LIN {X 0,Y 249.344,Z 174.923,A -85,B 0,C 180,E1 -18909.737,E2 -18909.737} C_VEL
LIN {X 0,Y 249.206,Z 174.945,A -85,B 0,C 180,E1 -18914.703,E2 -18914.703} C_VEL
LIN {X 0,Y 249.14,Z 174.944,A -85,B 0,C 180,E1 -18918.077,E2 -18918.077} C_VEL
LIN {X 0,Y 249.088,Z 174.954,A -85,B 0,C 180,E1 -18921.518,E2 -18921.518} C_VEL
LIN {X 0,Y 249.131,Z 174.951,A -85,B 0,C 180,E1 -18925.482,E2 -18925.482} C_VEL
LIN {X 0,Y 249.084,Z 174.957,A -85,B 0,C 180,E1 -18928.994,E2 -18928.994} C_VEL
LIN {X 0,Y 249.037,Z 174.96,A -85,B 0,C 180,E1 -18932.425,E2 -18932.425} C_VEL
LIN {X 0,Y 249.07,Z 174.957,A -85,B 0,C 180,E1 -18936.339,E2 -18936.339} C_VEL
LIN {X 0,Y 249.027,Z 174.966,A -85,B 0,C 180,E1 -18940.474,E2 -18940.474} C_VEL
LIN {X 0,Y 249.003,Z 174.965,A -85,B 0,C 180,E1 -18944.879,E2 -18944.879} C_VEL
LIN {X 0,Y 249.017,Z 174.965,A -85,B 0,C 180,E1 -18947.363,E2 -18947.363} C_VEL
LIN {X 0,Y 249.046,Z 174.962,A -85,B 0,C 180,E1 -18952.2,E2 -18952.2} C_VEL
LIN {X 0,Y 249.103,Z 175.108,A -85,B 0,C 180,E1 -18955.468,E2 -18955.468} C_VEL
LIN {X 0,Y 249.854,Z 178.125,A -85,B 0,C 180,E1 -18956.815,E2 -18956.815} C_VEL
LIN {X 0,Y 259.148,Z 197.045,A -85,B 0,C 180,E1 -18958.762,E2 -18958.762} C_VEL
LIN {X 0,Y 265.414,Z 211.933,A -85,B 0,C 180,E1 -18960.042,E2 -18960.042} C_VEL
LIN {X 0,Y 267.439,Z 217.922,A -85,B 0,C 180,E1 -18960.475,E2 -18960.475} C_VEL
LIN {X 0,Y 265.215,Z 283.423,A -85,B 0,C 180,E1 -18962.211,E2 -18962.211} C_VEL
LIN {X 0,Y 264.278,Z 296.661,A -85,B 0,C 180,E1 -18962.802,E2 -18962.802} C_VEL
LIN {X 0,Y 262.847,Z 309.804,A -85,B 0,C 180,E1 -18963.714,E2 -18963.714} C_VEL
LIN {X 0,Y 261.114,Z 322.253,A -85,B 0,C 180,E1 -18964.918,E2 -18964.918} C_VEL
LIN {X 0,Y 259.054,Z 333.896,A -85,B 0,C 180,E1 -18966.412,E2 -18966.412} C_VEL
LIN {X 0,Y 256.908,Z 344.67,A -85,B 0,C 180,E1 -18968.179,E2 -18968.179} C_VEL
LIN {X 0,Y 254.989,Z 354.577,A -85,B 0,C 180,E1 -18970.267,E2 -18970.267} C_VEL
LIN {X 0,Y 252.694,Z 363.495,A -85,B 0,C 180,E1 -18972.604,E2 -18972.604} C_VEL
LIN {X 0,Y 250.914,Z 370.67,A -85,B 0,C 180,E1 -18974.984,E2 -18974.984} C_VEL
LIN {X 0,Y 249.694,Z 375.507,A -85,B 0,C 180,E1 -18976.987,E2 -18976.987} C_VEL
LIN {X 0,Y 248.535,Z 380.207,A -85,B 0,C 180,E1 -18979.409,E2 -18979.409} C_VEL
LIN {X 0,Y 247.828,Z 383.8,A -85,B 0,C 180,E1 -18981.848,E2 -18981.848} C_VEL
LIN {X 0,Y 247.377,Z 386.053,A -85,B 0,C 180,E1 -18983.911,E2 -18983.911} C_VEL
LIN {X 0,Y 247.078,Z 388.044,A -85,B 0,C 180,E1 -18986.739,E2 -18986.739} C_VEL
LIN {X 0,Y 246.944,Z 388.884,A -85,B 0,C 180,E1 -18990,E2 -18990} C_VEL
LIN {X 0,Y 246.971,Z 388.691,A -85,B 0,C 180,E1 -18991.631,E2 -18991.631} C_VEL
LIN {X 0,Y 247.075,Z 388.104,A -85,B 0,C 180,E1 -18993.261,E2 -18993.261} C_VEL
LIN {X 0,Y 247.393,Z 385.779,A -85,B 0,C 180,E1 -18996.525,E2 -18996.525} C_VEL
LIN {X 0,Y 247.985,Z 382.908,A -85,B 0,C 180,E1 -18998.967,E2 -18998.967} C_VEL
LIN {X 0,Y 248.859,Z 379.014,A -85,B 0,C 180,E1 -19001.402,E2 -19001.402} C_VEL
LIN {X 0,Y 250.108,Z 373.989,A -85,B 0,C 180,E1 -19003.818,E2 -19003.818} C_VEL
LIN {X 0,Y 251.645,Z 367.662,A -85,B 0,C 180,E1 -19006.217,E2 -19006.217} C_VEL
LIN {X 0,Y 253.716,Z 359.739,A -85,B 0,C 180,E1 -19008.575,E2 -19008.575} C_VEL
LIN {X 0,Y 255.61,Z 351.261,A -85,B 0,C 180,E1 -19010.618,E2 -19010.618} C_VEL
LIN {X 0,Y 257.585,Z 341.814,A -85,B 0,C 180,E1 -19012.456,E2 -19012.456} C_VEL
LIN {X 0,Y 259.734,Z 330.721,A -85,B 0,C 180,E1 -19014.158,E2 -19014.158} C_VEL
LIN {X 0,Y 261.56,Z 319.844,A -85,B 0,C 180,E1 -19015.462,E2 -19015.462} C_VEL
LIN {X 0,Y 263.224,Z 307.822,A -85,B 0,C 180,E1 -19016.565,E2 -19016.565} C_VEL
LIN {X 0,Y 264.419,Z 295.46,A -85,B 0,C 180,E1 -19017.397,E2 -19017.397} C_VEL
LIN {X 0,Y 265.365,Z 282.621,A -85,B 0,C 180,E1 -19017.933,E2 -19017.933} C_VEL
LIN {X 0,Y 267.467,Z 217.517,A -85,B 0,C 180,E1 -19019.667,E2 -19019.667} C_VEL
LIN {X 0,Y 260.917,Z 200.918,A -85,B 0,C 180,E1 -19021.016,E2 -19021.016} C_VEL
LIN {X 0,Y 253.203,Z 184.855,A -85,B 0,C 180,E1 -19022.606,E2 -19022.606} C_VEL
LIN {X 0,Y 249.816,Z 177.906,A -85,B 0,C 180,E1 -19023.394,E2 -19023.394} C_VEL
LIN {X 0,Y 249.057,Z 174.953,A -85,B 0,C 180,E1 -19024.827,E2 -19024.827} C_VEL
LIN {X 0,Y 249.026,Z 174.967,A -85,B 0,C 180,E1 -19028.38,E2 -19028.38} C_VEL
LIN {X 0,Y 249.01,Z 174.968,A -85,B 0,C 180,E1 -19032.792,E2 -19032.792} C_VEL
LIN {X 0,Y 249.016,Z 174.965,A -85,B 0,C 180,E1 -19037.363,E2 -19037.363} C_VEL
LIN {X 0,Y 249.037,Z 174.959,A -85,B 0,C 180,E1 -19041.621,E2 -19041.621} C_VEL
LIN {X 0,Y 249.058,Z 174.956,A -85,B 0,C 180,E1 -19045.641,E2 -19045.641} C_VEL
LIN {X 0,Y 249.052,Z 174.962,A -85,B 0,C 180,E1 -19049.473,E2 -19049.473} C_VEL
LIN {X 0,Y 249.074,Z 174.953,A -85,B 0,C 180,E1 -19053.162,E2 -19053.162} C_VEL
LIN {X 0,Y 249.079,Z 174.954,A -85,B 0,C 180,E1 -19056.732,E2 -19056.732} C_VEL
LIN {X 0,Y 249.111,Z 174.953,A -85,B 0,C 180,E1 -19060.211,E2 -19060.211} C_VEL
LIN {X 0,Y 249.242,Z 174.927,A -85,B 0,C 180,E1 -19063.622,E2 -19063.622} C_VEL
LIN {X 0,Y 249.253,Z 174.937,A -85,B 0,C 180,E1 -19068.616,E2 -19068.616} C_VEL
LIN {X 0,Y 249.479,Z 174.897,A -85,B 0,C 180,E1 -19071.903,E2 -19071.903} C_VEL
LIN {X 0,Y 249.436,Z 174.911,A -85,B 0,C 180,E1 -19076.77,E2 -19076.77} C_VEL
LIN {X 0,Y 249.721,Z 174.87,A -85,B 0,C 180,E1 -19080,E2 -19080} C_VEL
LIN {X 0,Y 249.435,Z 174.912,A -85,B 0,C 180,E1 -19083.23,E2 -19083.23} C_VEL
LIN {X 0,Y 249.379,Z 174.907,A -85,B 0,C 180,E1 -19085.901,E2 -19085.901} C_VEL
LIN {X 0,Y 248.797,Z 174.987,A -85,B 0,C 180,E1 -19087.249,E2 -19087.249} C_VEL
LIN {X 0,Y 247.192,Z 175.192,A -85,B 0,C 180,E1 -19088.57,E2 -19088.57} C_VEL
LIN {X 0,Y 243.31,Z 175.672,A -85,B 0,C 180,E1 -19091.228,E2 -19091.228} C_VEL
LIN {X 0,Y 242.229,Z 175.8,A -85,B 0,C 180,E1 -19092.619,E2 -19092.619} C_VEL
LIN {X 0,Y 242.153,Z 175.807,A -85,B 0,C 180,E1 -19093.091,E2 -19093.091} C_VEL
LIN {X 0,Y 242.15,Z 175.819,A -85,B 0,C 180,E1 -19096.872,E2 -19096.872} C_VEL
LIN {X 0,Y 242.026,Z 175.834,A -85,B 0,C 180,E1 -19101.687,E2 -19101.687} C_VEL
LIN {X 0,Y 242.066,Z 175.824,A -85,B 0,C 180,E1 -19105.838,E2 -19105.838} C_VEL
LIN {X 0,Y 242.007,Z 175.835,A -85,B 0,C 180,E1 -19109.583,E2 -19109.583} C_VEL
LIN {X 0,Y 241.98,Z 175.841,A -85,B 0,C 180,E1 -19113.493,E2 -19113.493} C_VEL
LIN {X 0,Y 241.989,Z 175.839,A -85,B 0,C 180,E1 -19117.582,E2 -19117.582} C_VEL
LIN {X 0,Y 241.933,Z 175.846,A -85,B 0,C 180,E1 -19121.923,E2 -19121.923} C_VEL
LIN {X 0,Y 241.92,Z 175.85,A -85,B 0,C 180,E1 -19126.575,E2 -19126.575} C_VEL
LIN {X 0,Y 241.972,Z 176.038,A -85,B 0,C 180,E1 -19130.843,E2 -19130.843} C_VEL
LIN {X 0,Y 244.268,Z 184.837,A -85,B 0,C 180,E1 -19134.87,E2 -19134.87} C_VEL
LIN {X 0,Y 244.871,Z 187.317,A -85,B 0,C 180,E1 -19135.941,E2 -19135.941} C_VEL
LIN {X 0,Y 253.51,Z 206.311,A -85,B 0,C 180,E1 -19137.867,E2 -19137.867} C_VEL
LIN {X 0,Y 257.423,Z 216.174,A -85,B 0,C 180,E1 -19138.725,E2 -19138.725} C_VEL
LIN {X 0,Y 260.42,Z 235.313,A -85,B 0,C 180,E1 -19139.722,E2 -19139.722} C_VEL
LIN {X 0,Y 260.581,Z 240.387,A -85,B 0,C 180,E1 -19139.901,E2 -19139.901} C_VEL
LIN {X 0,Y 258.581,Z 296.119,A -85,B 0,C 180,E1 -19141.433,E2 -19141.433} C_VEL
LIN {X 0,Y 257.413,Z 309.243,A -85,B 0,C 180,E1 -19142.069,E2 -19142.069} C_VEL
LIN {X 0,Y 255.916,Z 321.325,A -85,B 0,C 180,E1 -19142.945,E2 -19142.945} C_VEL
LIN {X 0,Y 253.998,Z 333.525,A -85,B 0,C 180,E1 -19144.164,E2 -19144.164} C_VEL
LIN {X 0,Y 251.737,Z 345.085,A -85,B 0,C 180,E1 -19145.683,E2 -19145.683} C_VEL
LIN {X 0,Y 249.416,Z 355.496,A -85,B 0,C 180,E1 -19147.423,E2 -19147.423} C_VEL
LIN {X 0,Y 247.472,Z 364.011,A -85,B 0,C 180,E1 -19149.207,E2 -19149.207} C_VEL
LIN {X 0,Y 245.32,Z 373.244,A -85,B 0,C 180,E1 -19151.631,E2 -19151.631} C_VEL
LIN {X 0,Y 243.415,Z 380.664,A -85,B 0,C 180,E1 -19154.081,E2 -19154.081} C_VEL
LIN {X 0,Y 241.865,Z 386.623,A -85,B 0,C 180,E1 -19156.558,E2 -19156.558} C_VEL
LIN {X 0,Y 240.87,Z 391.336,A -85,B 0,C 180,E1 -19159.068,E2 -19159.068} C_VEL
LIN {X 0,Y 240.211,Z 394.938,A -85,B 0,C 180,E1 -19161.588,E2 -19161.588} C_VEL
LIN {X 0,Y 239.926,Z 396.795,A -85,B 0,C 180,E1 -19163.271,E2 -19163.271} C_VEL
LIN {X 0,Y 239.755,Z 399.185,A -85,B 0,C 180,E1 -19166.639,E2 -19166.639} C_VEL
LIN {X 0,Y 239.808,Z 399.793,A -85,B 0,C 180,E1 -19168.321,E2 -19168.321} C_VEL
LIN {X 0,Y 239.846,Z 400.005,A -85,B 0,C 180,E1 -19170,E2 -19170} C_VEL
LIN {X 0,Y 239.808,Z 399.782,A -85,B 0,C 180,E1 -19171.679,E2 -19171.679} C_VEL
LIN {X 0,Y 239.771,Z 398.373,A -85,B 0,C 180,E1 -19174.736,E2 -19174.736} C_VEL
LIN {X 0,Y 239.926,Z 396.76,A -85,B 0,C 180,E1 -19176.729,E2 -19176.729} C_VEL
LIN {X 0,Y 240.387,Z 393.815,A -85,B 0,C 180,E1 -19179.253,E2 -19179.253} C_VEL
LIN {X 0,Y 241.188,Z 389.833,A -85,B 0,C 180,E1 -19181.769,E2 -19181.769} C_VEL
LIN {X 0,Y 242.6,Z 383.713,A -85,B 0,C 180,E1 -19184.684,E2 -19184.684} C_VEL
LIN {X 0,Y 244.335,Z 377.034,A -85,B 0,C 180,E1 -19187.147,E2 -19187.147} C_VEL
LIN {X 0,Y 246.353,Z 368.317,A -85,B 0,C 180,E1 -19189.707,E2 -19189.707} C_VEL
LIN {X 0,Y 248.269,Z 360.245,A -85,B 0,C 180,E1 -19191.593,E2 -19191.593} C_VEL
LIN {X 0,Y 250.662,Z 349.747,A -85,B 0,C 180,E1 -19193.549,E2 -19193.549} C_VEL
LIN {X 0,Y 253.102,Z 337.93,A -85,B 0,C 180,E1 -19195.272,E2 -19195.272} C_VEL
LIN {X 0,Y 255.057,Z 326.019,A -85,B 0,C 180,E1 -19196.6,E2 -19196.6} C_VEL
LIN {X 0,Y 256.788,Z 313.622,A -85,B 0,C 180,E1 -19197.617,E2 -19197.617} C_VEL
LIN {X 0,Y 258.195,Z 300.844,A -85,B 0,C 180,E1 -19198.336,E2 -19198.336} C_VEL
LIN {X 0,Y 258.927,Z 287.293,A -85,B 0,C 180,E1 -19198.802,E2 -19198.802} C_VEL
LIN {X 0,Y 260.493,Z 236.282,A -85,B 0,C 180,E1 -19200.193,E2 -19200.193} C_VEL
LIN {X 0,Y 257.318,Z 215.805,A -85,B 0,C 180,E1 -19201.253,E2 -19201.253} C_VEL
LIN {X 0,Y 250.055,Z 198.58,A -85,B 0,C 180,E1 -19202.835,E2 -19202.835} C_VEL
LIN {X 0,Y 244.825,Z 187.196,A -85,B 0,C 180,E1 -19204.049,E2 -19204.049} C_VEL
LIN {X 0,Y 242.739,Z 178.842,A -85,B 0,C 180,E1 -19207.778,E2 -19207.778} C_VEL
LIN {X 0,Y 241.957,Z 175.847,A -85,B 0,C 180,E1 -19209.252,E2 -19209.252} C_VEL
LIN {X 0,Y 241.921,Z 175.851,A -85,B 0,C 180,E1 -19213.425,E2 -19213.425} C_VEL
LIN {X 0,Y 241.934,Z 175.849,A -85,B 0,C 180,E1 -19218.077,E2 -19218.077} C_VEL
LIN {X 0,Y 241.989,Z 175.842,A -85,B 0,C 180,E1 -19222.418,E2 -19222.418} C_VEL
LIN {X 0,Y 241.979,Z 175.844,A -85,B 0,C 180,E1 -19226.507,E2 -19226.507} C_VEL
LIN {X 0,Y 241.978,Z 175.843,A -85,B 0,C 180,E1 -19230.612,E2 -19230.612} C_VEL
LIN {X 0,Y 242.032,Z 175.836,A -85,B 0,C 180,E1 -19234.179,E2 -19234.179} C_VEL
LIN {X 0,Y 242.026,Z 175.835,A -85,B 0,C 180,E1 -19238.314,E2 -19238.314} C_VEL
LIN {X 0,Y 242.164,Z 175.814,A -85,B 0,C 180,E1 -19243.278,E2 -19243.278} C_VEL
LIN {X 0,Y 242.181,Z 175.812,A -85,B 0,C 180,E1 -19248.28,E2 -19248.28} C_VEL
LIN {X 0,Y 242.401,Z 175.788,A -85,B 0,C 180,E1 -19251.665,E2 -19251.665} C_VEL
LIN {X 0,Y 242.257,Z 175.804,A -85,B 0,C 180,E1 -19255.007,E2 -19255.007} C_VEL
LIN {X 0,Y 242.637,Z 175.756,A -85,B 0,C 180,E1 -19258.34,E2 -19258.34} C_VEL
LIN {X 0,Y 242.636,Z 175.761,A -85,B 0,C 180,E1 -19261.66,E2 -19261.66} C_VEL
LIN {X 0,Y 242.423,Z 175.781,A -85,B 0,C 180,E1 -19266.659,E2 -19266.659} C_VEL
LIN {X 0,Y 242.268,Z 175.804,A -85,B 0,C 180,E1 -19270.024,E2 -19270.024} C_VEL
LIN {X 0,Y 242.167,Z 175.818,A -85,B 0,C 180,E1 -19275.141,E2 -19275.141} C_VEL
LIN {X 0,Y 242.074,Z 175.827,A -85,B 0,C 180,E1 -19278.624,E2 -19278.624} C_VEL
LIN {X 0,Y 242.014,Z 175.833,A -85,B 0,C 180,E1 -19282.18,E2 -19282.18} C_VEL
LIN {X 0,Y 242.067,Z 175.831,A -85,B 0,C 180,E1 -19285.838,E2 -19285.838} C_VEL
LIN {X 0,Y 242.031,Z 175.835,A -85,B 0,C 180,E1 -19289.58,E2 -19289.58} C_VEL
LIN {X 0,Y 241.992,Z 175.84,A -85,B 0,C 180,E1 -19293.491,E2 -19293.491} C_VEL
LIN {X 0,Y 242.003,Z 175.84,A -85,B 0,C 180,E1 -19297.58,E2 -19297.58} C_VEL
LIN {X 0,Y 241.944,Z 175.846,A -85,B 0,C 180,E1 -19301.921,E2 -19301.921} C_VEL
LIN {X 0,Y 241.935,Z 175.847,A -85,B 0,C 180,E1 -19306.571,E2 -19306.571} C_VEL
LIN {X 0,Y 241.958,Z 175.844,A -85,B 0,C 180,E1 -19310.281,E2 -19310.281} C_VEL
LIN {X 0,Y 242.02,Z 175.849,A -85,B 0,C 180,E1 -19314.546,E2 -19314.546} C_VEL
LIN {X 0,Y 242.628,Z 178.345,A -85,B 0,C 180,E1 -19315.691,E2 -19315.691} C_VEL
LIN {X 0,Y 251.925,Z 196.7,A -85,B 0,C 180,E1 -19317.741,E2 -19317.741} C_VEL
LIN {X 0,Y 258.644,Z 212.335,A -85,B 0,C 180,E1 -19319.18,E2 -19319.18} C_VEL
LIN {X 0,Y 261.151,Z 219.015,A -85,B 0,C 180,E1 -19319.719,E2 -19319.719} C_VEL
LIN {X 0,Y 259.029,Z 282.511,A -85,B 0,C 180,E1 -19321.447,E2 -19321.447} C_VEL
LIN {X 0,Y 258.152,Z 295.304,A -85,B 0,C 180,E1 -19321.996,E2 -19321.996} C_VEL
LIN {X 0,Y 256.799,Z 307.717,A -85,B 0,C 180,E1 -19322.826,E2 -19322.826} C_VEL
LIN {X 0,Y 254.972,Z 320.685,A -85,B 0,C 180,E1 -19324.051,E2 -19324.051} C_VEL
LIN {X 0,Y 253.06,Z 331.432,A -85,B 0,C 180,E1 -19325.381,E2 -19325.381} C_VEL
LIN {X 0,Y 250.823,Z 342.491,A -85,B 0,C 180,E1 -19327.144,E2 -19327.144} C_VEL
LIN {X 0,Y 248.865,Z 351.996,A -85,B 0,C 180,E1 -19329.071,E2 -19329.071} C_VEL
LIN {X 0,Y 246.654,Z 360.923,A -85,B 0,C 180,E1 -19331.304,E2 -19331.304} C_VEL
LIN {X 0,Y 244.597,Z 368.613,A -85,B 0,C 180,E1 -19333.731,E2 -19333.731} C_VEL
LIN {X 0,Y 242.762,Z 375.671,A -85,B 0,C 180,E1 -19336.609,E2 -19336.609} C_VEL
LIN {X 0,Y 241.553,Z 380.37,A -85,B 0,C 180,E1 -19339.099,E2 -19339.099} C_VEL
LIN {X 0,Y 240.789,Z 383.963,A -85,B 0,C 180,E1 -19341.608,E2 -19341.608} C_VEL
LIN {X 0,Y 240.287,Z 386.411,A -85,B 0,C 180,E1 -19343.96,E2 -19343.96} C_VEL
LIN {X 0,Y 240.002,Z 388.206,A -85,B 0,C 180,E1 -19346.642,E2 -19346.642} C_VEL
LIN {X 0,Y 239.855,Z 389.046,A -85,B 0,C 180,E1 -19350,E2 -19350} C_VEL
LIN {X 0,Y 239.886,Z 388.853,A -85,B 0,C 180,E1 -19351.679,E2 -19351.679} C_VEL
LIN {X 0,Y 239.997,Z 388.266,A -85,B 0,C 180,E1 -19353.357,E2 -19353.357} C_VEL
LIN {X 0,Y 240.349,Z 385.941,A -85,B 0,C 180,E1 -19356.717,E2 -19356.717} C_VEL
LIN {X 0,Y 240.972,Z 383.069,A -85,B 0,C 180,E1 -19359.23,E2 -19359.23} C_VEL
LIN {X 0,Y 241.897,Z 379.175,A -85,B 0,C 180,E1 -19361.734,E2 -19361.734} C_VEL
LIN {X 0,Y 243.217,Z 374.15,A -85,B 0,C 180,E1 -19364.218,E2 -19364.218} C_VEL
LIN {X 0,Y 244.831,Z 367.822,A -85,B 0,C 180,E1 -19366.682,E2 -19366.682} C_VEL
LIN {X 0,Y 246.999,Z 359.899,A -85,B 0,C 180,E1 -19369.1,E2 -19369.1} C_VEL
LIN {X 0,Y 248.824,Z 352.038,A -85,B 0,C 180,E1 -19371.056,E2 -19371.056} C_VEL
LIN {X 0,Y 251.03,Z 341.973,A -85,B 0,C 180,E1 -19373.076,E2 -19373.076} C_VEL
LIN {X 0,Y 253.291,Z 330.878,A -85,B 0,C 180,E1 -19374.814,E2 -19374.814} C_VEL
LIN {X 0,Y 255.174,Z 320,A -85,B 0,C 180,E1 -19376.147,E2 -19376.147} C_VEL
LIN {X 0,Y 256.908,Z 307.976,A -85,B 0,C 180,E1 -19377.272,E2 -19377.272} C_VEL
LIN {X 0,Y 258.138,Z 295.611,A -85,B 0,C 180,E1 -19378.121,E2 -19378.121} C_VEL
LIN {X 0,Y 259.125,Z 282.763,A -85,B 0,C 180,E1 -19378.667,E2 -19378.667} C_VEL
LIN {X 0,Y 261.284,Z 219.256,A -85,B 0,C 180,E1 -19380.392,E2 -19380.392} C_VEL
LIN {X 0,Y 255.424,Z 204.408,A -85,B 0,C 180,E1 -19381.65,E2 -19381.65} C_VEL
LIN {X 0,Y 248.107,Z 188.989,A -85,B 0,C 180,E1 -19383.225,E2 -19383.225} C_VEL
LIN {X 0,Y 243.691,Z 180.673,A -85,B 0,C 180,E1 -19384.202,E2 -19384.202} C_VEL
LIN {X 0,Y 242.589,Z 178.173,A -85,B 0,C 180,E1 -19384.494,E2 -19384.494} C_VEL
LIN {X 0,Y 242.01,Z 175.835,A -85,B 0,C 180,E1 -19385.666,E2 -19385.666} C_VEL
LIN {X 0,Y 241.957,Z 175.843,A -85,B 0,C 180,E1 -19389.719,E2 -19389.719} C_VEL
LIN {X 0,Y 241.931,Z 175.847,A -85,B 0,C 180,E1 -19394.202,E2 -19394.202} C_VEL
LIN {X 0,Y 241.943,Z 175.843,A -85,B 0,C 180,E1 -19398.079,E2 -19398.079} C_VEL
LIN {X 0,Y 241.999,Z 175.834,A -85,B 0,C 180,E1 -19402.42,E2 -19402.42} C_VEL
LIN {X 0,Y 241.989,Z 175.831,A -85,B 0,C 180,E1 -19406.508,E2 -19406.508} C_VEL
LIN {X 0,Y 242.037,Z 175.831,A -85,B 0,C 180,E1 -19410.587,E2 -19410.587} C_VEL
LIN {X 0,Y 242.068,Z 175.832,A -85,B 0,C 180,E1 -19414.183,E2 -19414.183} C_VEL
LIN {X 0,Y 242.053,Z 175.824,A -85,B 0,C 180,E1 -19418.297,E2 -19418.297} C_VEL
LIN {X 0,Y 242.163,Z 175.811,A -85,B 0,C 180,E1 -19423.278,E2 -19423.278} C_VEL
LIN {X 0,Y 242.186,Z 175.816,A -85,B 0,C 180,E1 -19428.28,E2 -19428.28} C_VEL
LIN {X 0,Y 242.426,Z 175.774,A -85,B 0,C 180,E1 -19431.665,E2 -19431.665} C_VEL
LIN {X 0,Y 242.259,Z 175.81,A -85,B 0,C 180,E1 -19435.007,E2 -19435.007} C_VEL
LIN {X 0,Y 242.636,Z 175.749,A -85,B 0,C 180,E1 -19438.34,E2 -19438.34} C_VEL
LIN {X 0,Y 242.636,Z 175.76,A -85,B 0,C 180,E1 -19441.66,E2 -19441.66} C_VEL
LIN {X 0,Y 242.431,Z 175.774,A -85,B 0,C 180,E1 -19446.659,E2 -19446.659} C_VEL
LIN {X 0,Y 242.314,Z 175.801,A -85,B 0,C 180,E1 -19450.022,E2 -19450.022} C_VEL
LIN {X 0,Y 242.153,Z 175.807,A -85,B 0,C 180,E1 -19453.091,E2 -19453.091} C_VEL
LIN {X 0,Y 241.497,Z 175.897,A -85,B 0,C 180,E1 -19454.479,E2 -19454.479} C_VEL
LIN {X 0,Y 238.58,Z 176.265,A -85,B 0,C 180,E1 -19456.739,E2 -19456.739} C_VEL
LIN {X 0,Y 236.097,Z 176.566,A -85,B 0,C 180,E1 -19458.582,E2 -19458.582} C_VEL
LIN {X 0,Y 235.05,Z 176.694,A -85,B 0,C 180,E1 -19460.015,E2 -19460.015} C_VEL
LIN {X 0,Y 234.975,Z 176.706,A -85,B 0,C 180,E1 -19460.501,E2 -19460.501} C_VEL
LIN {X 0,Y 234.977,Z 176.705,A -85,B 0,C 180,E1 -19464.754,E2 -19464.754} C_VEL
LIN {X 0,Y 234.936,Z 176.718,A -85,B 0,C 180,E1 -19468.596,E2 -19468.596} C_VEL
LIN {X 0,Y 234.942,Z 176.719,A -85,B 0,C 180,E1 -19473.115,E2 -19473.115} C_VEL
LIN {X 0,Y 234.927,Z 176.721,A -85,B 0,C 180,E1 -19476.749,E2 -19476.749} C_VEL
LIN {X 0,Y 234.942,Z 176.716,A -85,B 0,C 180,E1 -19478.945,E2 -19478.945} C_VEL
LIN {X 0,Y 234.878,Z 176.727,A -85,B 0,C 180,E1 -19483.488,E2 -19483.488} C_VEL
LIN {X 0,Y 234.873,Z 176.727,A -85,B 0,C 180,E1 -19486.511,E2 -19486.511} C_VEL
LIN {X 0,Y 234.903,Z 176.735,A -85,B 0,C 180,E1 -19489.826,E2 -19489.826} C_VEL
LIN {X 0,Y 236.976,Z 184.637,A -85,B 0,C 180,E1 -19493.62,E2 -19493.62} C_VEL
LIN {X 0,Y 237.564,Z 187.033,A -85,B 0,C 180,E1 -19494.717,E2 -19494.717} C_VEL
LIN {X 0,Y 245.781,Z 204.508,A -85,B 0,C 180,E1 -19496.673,E2 -19496.673} C_VEL
LIN {X 0,Y 251.518,Z 218.485,A -85,B 0,C 180,E1 -19497.985,E2 -19497.985} C_VEL
LIN {X 0,Y 254.367,Z 236.86,A -85,B 0,C 180,E1 -19498.977,E2 -19498.977} C_VEL
LIN {X 0,Y 254.306,Z 245.216,A -85,B 0,C 180,E1 -19499.238,E2 -19499.238} C_VEL
LIN {X 0,Y 252.374,Z 295.97,A -85,B 0,C 180,E1 -19500.663,E2 -19500.663} C_VEL
LIN {X 0,Y 251.178,Z 309.09,A -85,B 0,C 180,E1 -19501.313,E2 -19501.313} C_VEL
LIN {X 0,Y 249.595,Z 321.169,A -85,B 0,C 180,E1 -19502.202,E2 -19502.202} C_VEL
LIN {X 0,Y 247.634,Z 333.368,A -85,B 0,C 180,E1 -19503.449,E2 -19503.449} C_VEL
LIN {X 0,Y 245.276,Z 344.927,A -85,B 0,C 180,E1 -19504.999,E2 -19504.999} C_VEL
LIN {X 0,Y 242.866,Z 355.337,A -85,B 0,C 180,E1 -19506.779,E2 -19506.779} C_VEL
LIN {X 0,Y 240.82,Z 363.851,A -85,B 0,C 180,E1 -19508.605,E2 -19508.605} C_VEL
LIN {X 0,Y 239.038,Z 371.442,A -85,B 0,C 180,E1 -19510.604,E2 -19510.604} C_VEL
LIN {X 0,Y 236.906,Z 379.383,A -85,B 0,C 180,E1 -19513.188,E2 -19513.188} C_VEL
LIN {X 0,Y 234.926,Z 386.461,A -85,B 0,C 180,E1 -19516.153,E2 -19516.153} C_VEL
LIN {X 0,Y 233.887,Z 391.174,A -85,B 0,C 180,E1 -19518.737,E2 -19518.737} C_VEL
LIN {X 0,Y 233.179,Z 394.776,A -85,B 0,C 180,E1 -19521.333,E2 -19521.333} C_VEL
LIN {X 0,Y 232.872,Z 396.633,A -85,B 0,C 180,E1 -19523.067,E2 -19523.067} C_VEL
LIN {X 0,Y 232.666,Z 399.023,A -85,B 0,C 180,E1 -19526.537,E2 -19526.537} C_VEL
LIN {X 0,Y 232.722,Z 399.631,A -85,B 0,C 180,E1 -19528.27,E2 -19528.27} C_VEL
LIN {X 0,Y 232.759,Z 399.844,A -85,B 0,C 180,E1 -19530,E2 -19530} C_VEL
LIN {X 0,Y 232.722,Z 399.62,A -85,B 0,C 180,E1 -19531.731,E2 -19531.731} C_VEL
LIN {X 0,Y 232.73,Z 398.003,A -85,B 0,C 180,E1 -19535.198,E2 -19535.198} C_VEL
LIN {X 0,Y 232.872,Z 396.597,A -85,B 0,C 180,E1 -19536.934,E2 -19536.934} C_VEL
LIN {X 0,Y 233.372,Z 393.652,A -85,B 0,C 180,E1 -19539.534,E2 -19539.534} C_VEL
LIN {X 0,Y 234.223,Z 389.67,A -85,B 0,C 180,E1 -19542.125,E2 -19542.125} C_VEL
LIN {X 0,Y 235.725,Z 383.549,A -85,B 0,C 180,E1 -19545.122,E2 -19545.122} C_VEL
LIN {X 0,Y 237.496,Z 376.868,A -85,B 0,C 180,E1 -19547.657,E2 -19547.657} C_VEL
LIN {X 0,Y 239.496,Z 368.781,A -85,B 0,C 180,E1 -19550.109,E2 -19550.109} C_VEL
LIN {X 0,Y 241.662,Z 360.079,A -85,B 0,C 180,E1 -19552.214,E2 -19552.214} C_VEL
LIN {X 0,Y 244.169,Z 349.581,A -85,B 0,C 180,E1 -19554.215,E2 -19554.215} C_VEL
LIN {X 0,Y 246.685,Z 337.763,A -85,B 0,C 180,E1 -19555.978,E2 -19555.978} C_VEL
LIN {X 0,Y 248.724,Z 325.85,A -85,B 0,C 180,E1 -19557.333,E2 -19557.333} C_VEL
LIN {X 0,Y 250.534,Z 313.453,A -85,B 0,C 180,E1 -19558.368,E2 -19558.368} C_VEL
LIN {X 0,Y 251.981,Z 300.67,A -85,B 0,C 180,E1 -19559.101,E2 -19559.101} C_VEL
LIN {X 0,Y 252.736,Z 287.109,A -85,B 0,C 180,E1 -19559.576,E2 -19559.576} C_VEL
LIN {X 0,Y 254.368,Z 237.436,A -85,B 0,C 180,E1 -19560.956,E2 -19560.956} C_VEL
LIN {X 0,Y 251.342,Z 218.086,A -85,B 0,C 180,E1 -19562.003,E2 -19562.003} C_VEL
LIN {X 0,Y 244.397,Z 201.525,A -85,B 0,C 180,E1 -19563.588,E2 -19563.588} C_VEL
LIN {X 0,Y 239.171,Z 190.512,A -85,B 0,C 180,E1 -19564.81,E2 -19564.81} C_VEL
LIN {X 0,Y 237.55,Z 186.991,A -85,B 0,C 180,E1 -19565.245,E2 -19565.245} C_VEL
LIN {X 0,Y 235.442,Z 178.8,A -85,B 0,C 180,E1 -19569.094,E2 -19569.094} C_VEL
LIN {X 0,Y 234.904,Z 176.727,A -85,B 0,C 180,E1 -19570.174,E2 -19570.174} C_VEL
LIN {X 0,Y 234.882,Z 176.729,A -85,B 0,C 180,E1 -19574.101,E2 -19574.101} C_VEL
LIN {X 0,Y 234.882,Z 176.727,A -85,B 0,C 180,E1 -19578.832,E2 -19578.832} C_VEL
LIN {X 0,Y 234.918,Z 176.723,A -85,B 0,C 180,E1 -19581.079,E2 -19581.079} C_VEL
LIN {X 0,Y 234.93,Z 176.72,A -85,B 0,C 180,E1 -19585.362,E2 -19585.362} C_VEL
LIN {X 0,Y 234.899,Z 176.724,A -85,B 0,C 180,E1 -19589.428,E2 -19589.428} C_VEL
LIN {X 0,Y 234.969,Z 176.713,A -85,B 0,C 180,E1 -19593.806,E2 -19593.806} C_VEL
LIN {X 0,Y 234.998,Z 176.711,A -85,B 0,C 180,E1 -19598.969,E2 -19598.969} C_VEL
LIN {X 0,Y 235.097,Z 176.694,A -85,B 0,C 180,E1 -19603.06,E2 -19603.06} C_VEL
LIN {X 0,Y 235.115,Z 176.69,A -85,B 0,C 180,E1 -19607.922,E2 -19607.922} C_VEL
LIN {X 0,Y 235.332,Z 176.671,A -85,B 0,C 180,E1 -19611.412,E2 -19611.412} C_VEL
LIN {X 0,Y 235.374,Z 176.658,A -85,B 0,C 180,E1 -19613.141,E2 -19613.141} C_VEL
LIN {X 0,Y 235.596,Z 176.633,A -85,B 0,C 180,E1 -19618.291,E2 -19618.291} C_VEL
LIN {X 0,Y 235.596,Z 176.638,A -85,B 0,C 180,E1 -19621.71,E2 -19621.71} C_VEL
LIN {X 0,Y 235.373,Z 176.66,A -85,B 0,C 180,E1 -19626.86,E2 -19626.86} C_VEL
LIN {X 0,Y 235.215,Z 176.683,A -85,B 0,C 180,E1 -19630.328,E2 -19630.328} C_VEL
LIN {X 0,Y 235.114,Z 176.695,A -85,B 0,C 180,E1 -19635.606,E2 -19635.606} C_VEL
LIN {X 0,Y 235.01,Z 176.711,A -85,B 0,C 180,E1 -19639.206,E2 -19639.206} C_VEL
LIN {X 0,Y 234.962,Z 176.71,A -85,B 0,C 180,E1 -19642.883,E2 -19642.883} C_VEL
LIN {X 0,Y 234.97,Z 176.711,A -85,B 0,C 180,E1 -19646.657,E2 -19646.657} C_VEL
LIN {X 0,Y 234.933,Z 176.719,A -85,B 0,C 180,E1 -19650.568,E2 -19650.568} C_VEL
LIN {X 0,Y 234.961,Z 176.716,A -85,B 0,C 180,E1 -19654.633,E2 -19654.633} C_VEL
LIN {X 0,Y 234.943,Z 176.716,A -85,B 0,C 180,E1 -19658.945,E2 -19658.945} C_VEL
LIN {X 0,Y 234.888,Z 176.725,A -85,B 0,C 180,E1 -19663.486,E2 -19663.486} C_VEL
LIN {X 0,Y 234.888,Z 176.725,A -85,B 0,C 180,E1 -19666.514,E2 -19666.514} C_VEL
LIN {X 0,Y 234.92,Z 176.723,A -85,B 0,C 180,E1 -19671.079,E2 -19671.079} C_VEL
LIN {X 0,Y 234.945,Z 176.766,A -85,B 0,C 180,E1 -19673.637,E2 -19673.637} C_VEL
LIN {X 0,Y 235.422,Z 178.477,A -85,B 0,C 180,E1 -19674.482,E2 -19674.482} C_VEL
LIN {X 0,Y 243.963,Z 195.042,A -85,B 0,C 180,E1 -19676.487,E2 -19676.487} C_VEL
LIN {X 0,Y 250.222,Z 208.547,A -85,B 0,C 180,E1 -19677.888,E2 -19677.888} C_VEL
LIN {X 0,Y 255.041,Z 220.804,A -85,B 0,C 180,E1 -19678.966,E2 -19678.966} C_VEL
LIN {X 0,Y 252.771,Z 283.588,A -85,B 0,C 180,E1 -19680.706,E2 -19680.706} C_VEL
LIN {X 0,Y 251.822,Z 296.475,A -85,B 0,C 180,E1 -19681.296,E2 -19681.296} C_VEL
LIN {X 0,Y 250.372,Z 309.015,A -85,B 0,C 180,E1 -19682.182,E2 -19682.182} C_VEL
LIN {X 0,Y 248.624,Z 320.853,A -85,B 0,C 180,E1 -19683.337,E2 -19683.337} C_VEL
LIN {X 0,Y 246.622,Z 331.599,A -85,B 0,C 180,E1 -19684.694,E2 -19684.694} C_VEL
LIN {X 0,Y 244.291,Z 342.657,A -85,B 0,C 180,E1 -19686.496,E2 -19686.496} C_VEL
LIN {X 0,Y 242.135,Z 352.592,A -85,B 0,C 180,E1 -19688.569,E2 -19688.569} C_VEL
LIN {X 0,Y 239.947,Z 361.087,A -85,B 0,C 180,E1 -19690.761,E2 -19690.761} C_VEL
LIN {X 0,Y 237.792,Z 368.777,A -85,B 0,C 180,E1 -19693.252,E2 -19693.252} C_VEL
LIN {X 0,Y 235.853,Z 375.835,A -85,B 0,C 180,E1 -19696.209,E2 -19696.209} C_VEL
LIN {X 0,Y 234.589,Z 380.534,A -85,B 0,C 180,E1 -19698.771,E2 -19698.771} C_VEL
LIN {X 0,Y 233.746,Z 384.127,A -85,B 0,C 180,E1 -19701.354,E2 -19701.354} C_VEL
LIN {X 0,Y 233.18,Z 386.804,A -85,B 0,C 180,E1 -19704.053,E2 -19704.053} C_VEL
LIN {X 0,Y 232.908,Z 388.369,A -85,B 0,C 180,E1 -19706.54,E2 -19706.54} C_VEL
LIN {X 0,Y 232.804,Z 388.979,A -85,B 0,C 180,E1 -19708.27,E2 -19708.27} C_VEL
LIN {X 0,Y 232.768,Z 389.208,A -85,B 0,C 180,E1 -19710,E2 -19710} C_VEL
LIN {X 0,Y 232.803,Z 389.015,A -85,B 0,C 180,E1 -19711.73,E2 -19711.73} C_VEL
LIN {X 0,Y 232.902,Z 388.428,A -85,B 0,C 180,E1 -19713.46,E2 -19713.46} C_VEL
LIN {X 0,Y 233.3,Z 386.102,A -85,B 0,C 180,E1 -19716.921,E2 -19716.921} C_VEL
LIN {X 0,Y 233.959,Z 383.231,A -85,B 0,C 180,E1 -19719.51,E2 -19719.51} C_VEL
LIN {X 0,Y 234.95,Z 379.336,A -85,B 0,C 180,E1 -19722.086,E2 -19722.086} C_VEL
LIN {X 0,Y 236.339,Z 374.31,A -85,B 0,C 180,E1 -19724.641,E2 -19724.641} C_VEL
LIN {X 0,Y 238.043,Z 367.982,A -85,B 0,C 180,E1 -19727.172,E2 -19727.172} C_VEL
LIN {X 0,Y 240.304,Z 360.058,A -85,B 0,C 180,E1 -19729.653,E2 -19729.653} C_VEL
LIN {X 0,Y 242.5,Z 350.876,A -85,B 0,C 180,E1 -19731.965,E2 -19731.965} C_VEL
LIN {X 0,Y 244.777,Z 341.032,A -85,B 0,C 180,E1 -19733.926,E2 -19733.926} C_VEL
LIN {X 0,Y 246.865,Z 331.035,A -85,B 0,C 180,E1 -19735.505,E2 -19735.505} C_VEL
LIN {X 0,Y 248.84,Z 320.156,A -85,B 0,C 180,E1 -19736.865,E2 -19736.865} C_VEL
LIN {X 0,Y 250.632,Z 308.13,A -85,B 0,C 180,E1 -19738.014,E2 -19738.014} C_VEL
LIN {X 0,Y 251.914,Z 295.761,A -85,B 0,C 180,E1 -19738.881,E2 -19738.881} C_VEL
LIN {X 0,Y 252.916,Z 282.905,A -85,B 0,C 180,E1 -19739.439,E2 -19739.439} C_VEL
LIN {X 0,Y 255.143,Z 221.008,A -85,B 0,C 180,E1 -19741.152,E2 -19741.152} C_VEL
LIN {X 0,Y 249.505,Z 206.754,A -85,B 0,C 180,E1 -19742.418,E2 -19742.418} C_VEL
LIN {X 0,Y 242.527,Z 192.121,A -85,B 0,C 180,E1 -19743.988,E2 -19743.988} C_VEL
LIN {X 0,Y 236.929,Z 181.571,A -85,B 0,C 180,E1 -19745.294,E2 -19745.294} C_VEL
LIN {X 0,Y 235.364,Z 178.311,A -85,B 0,C 180,E1 -19745.737,E2 -19745.737} C_VEL
LIN {X 0,Y 234.983,Z 176.715,A -85,B 0,C 180,E1 -19746.549,E2 -19746.549} C_VEL
LIN {X 0,Y 234.943,Z 176.718,A -85,B 0,C 180,E1 -19748.944,E2 -19748.944} C_VEL
LIN {X 0,Y 234.888,Z 176.727,A -85,B 0,C 180,E1 -19753.486,E2 -19753.486} C_VEL
LIN {X 0,Y 234.888,Z 176.727,A -85,B 0,C 180,E1 -19756.514,E2 -19756.514} C_VEL
LIN {X 0,Y 234.955,Z 176.715,A -85,B 0,C 180,E1 -19761.086,E2 -19761.086} C_VEL
LIN {X 0,Y 234.96,Z 176.714,A -85,B 0,C 180,E1 -19765.367,E2 -19765.367} C_VEL
LIN {X 0,Y 234.97,Z 176.713,A -85,B 0,C 180,E1 -19770.157,E2 -19770.157} C_VEL
LIN {X 0,Y 234.994,Z 176.711,A -85,B 0,C 180,E1 -19773.793,E2 -19773.793} C_VEL
LIN {X 0,Y 235.012,Z 176.702,A -85,B 0,C 180,E1 -19778.97,E2 -19778.97} C_VEL
LIN {X 0,Y 235.096,Z 176.693,A -85,B 0,C 180,E1 -19783.059,E2 -19783.059} C_VEL
LIN {X 0,Y 235.147,Z 176.693,A -85,B 0,C 180,E1 -19787.924,E2 -19787.924} C_VEL
LIN {X 0,Y 235.376,Z 176.651,A -85,B 0,C 180,E1 -19791.414,E2 -19791.414} C_VEL
LIN {X 0,Y 235.402,Z 176.655,A -85,B 0,C 180,E1 -19793.141,E2 -19793.141} C_VEL
LIN {X 0,Y 235.596,Z 176.625,A -85,B 0,C 180,E1 -19798.29,E2 -19798.29} C_VEL
LIN {X 0,Y 235.596,Z 176.637,A -85,B 0,C 180,E1 -19801.709,E2 -19801.709} C_VEL
LIN {X 0,Y 235.402,Z 176.65,A -85,B 0,C 180,E1 -19806.859,E2 -19806.859} C_VEL
LIN {X 0,Y 235.238,Z 176.683,A -85,B 0,C 180,E1 -19810.326,E2 -19810.326} C_VEL
LIN {X 0,Y 235.113,Z 176.695,A -85,B 0,C 180,E1 -19815.606,E2 -19815.606} C_VEL
LIN {X 0,Y 235.007,Z 176.699,A -85,B 0,C 180,E1 -19819.206,E2 -19819.206} C_VEL
LIN {X 0,Y 234.975,Z 176.706,A -85,B 0,C 180,E1 -19820.501,E2 -19820.501} C_VEL
LIN {X 0,Y 234.331,Z 176.796,A -85,B 0,C 180,E1 -19821.932,E2 -19821.932} C_VEL
LIN {X 0,Y 231.467,Z 177.161,A -85,B 0,C 180,E1 -19824.265,E2 -19824.265} C_VEL
LIN {X 0,Y 229.009,Z 177.463,A -85,B 0,C 180,E1 -19826.168,E2 -19826.168} C_VEL
LIN {X 0,Y 227.947,Z 177.591,A -85,B 0,C 180,E1 -19827.646,E2 -19827.646} C_VEL
LIN {X 0,Y 227.857,Z 177.597,A -85,B 0,C 180,E1 -19828.148,E2 -19828.148} C_VEL
LIN {X 0,Y 227.866,Z 177.598,A -85,B 0,C 180,E1 -19831.623,E2 -19831.623} C_VEL
LIN {X 0,Y 227.881,Z 177.598,A -85,B 0,C 180,E1 -19835.872,E2 -19835.872} C_VEL
LIN {X 0,Y 227.824,Z 177.606,A -85,B 0,C 180,E1 -19840.377,E2 -19840.377} C_VEL
LIN {X 0,Y 227.824,Z 177.605,A -85,B 0,C 180,E1 -19845.195,E2 -19845.195} C_VEL
LIN {X 0,Y 227.847,Z 177.693,A -85,B 0,C 180,E1 -19848.856,E2 -19848.856} C_VEL
LIN {X 0,Y 230.26,Z 186.82,A -85,B 0,C 180,E1 -19853.415,E2 -19853.415} C_VEL
LIN {X 0,Y 238.305,Z 203.256,A -85,B 0,C 180,E1 -19855.444,E2 -19855.444} C_VEL
LIN {X 0,Y 244.848,Z 218.78,A -85,B 0,C 180,E1 -19857.019,E2 -19857.019} C_VEL
LIN {X 0,Y 246.098,Z 222.895,A -85,B 0,C 180,E1 -19857.347,E2 -19857.347} C_VEL
LIN {X 0,Y 248.428,Z 239.786,A -85,B 0,C 180,E1 -19858.252,E2 -19858.252} C_VEL
LIN {X 0,Y 246.214,Z 295.822,A -85,B 0,C 180,E1 -19859.855,E2 -19859.855} C_VEL
LIN {X 0,Y 244.985,Z 308.937,A -85,B 0,C 180,E1 -19860.517,E2 -19860.517} C_VEL
LIN {X 0,Y 243.337,Z 321.014,A -85,B 0,C 180,E1 -19861.422,E2 -19861.422} C_VEL
LIN {X 0,Y 241.311,Z 333.211,A -85,B 0,C 180,E1 -19862.697,E2 -19862.697} C_VEL
LIN {X 0,Y 238.866,Z 344.769,A -85,B 0,C 180,E1 -19864.28,E2 -19864.28} C_VEL
LIN {X 0,Y 236.335,Z 355.177,A -85,B 0,C 180,E1 -19866.098,E2 -19866.098} C_VEL
LIN {X 0,Y 234.189,Z 363.69,A -85,B 0,C 180,E1 -19867.968,E2 -19867.968} C_VEL
LIN {X 0,Y 231.841,Z 372.923,A -85,B 0,C 180,E1 -19870.522,E2 -19870.522} C_VEL
LIN {X 0,Y 229.77,Z 380.342,A -85,B 0,C 180,E1 -19873.108,E2 -19873.108} C_VEL
LIN {X 0,Y 228.008,Z 386.3,A -85,B 0,C 180,E1 -19875.724,E2 -19875.724} C_VEL
LIN {X 0,Y 226.899,Z 391.013,A -85,B 0,C 180,E1 -19878.385,E2 -19878.385} C_VEL
LIN {X 0,Y 226.138,Z 394.614,A -85,B 0,C 180,E1 -19881.061,E2 -19881.061} C_VEL
LIN {X 0,Y 225.809,Z 396.471,A -85,B 0,C 180,E1 -19882.849,E2 -19882.849} C_VEL
LIN {X 0,Y 225.581,Z 398.861,A -85,B 0,C 180,E1 -19886.428,E2 -19886.428} C_VEL
LIN {X 0,Y 225.618,Z 399.469,A -85,B 0,C 180,E1 -19888.215,E2 -19888.215} C_VEL
LIN {X 0,Y 225.674,Z 399.682,A -85,B 0,C 180,E1 -19890,E2 -19890} C_VEL
LIN {X 0,Y 225.618,Z 399.457,A -85,B 0,C 180,E1 -19891.785,E2 -19891.785} C_VEL
LIN {X 0,Y 225.584,Z 398.402,A -85,B 0,C 180,E1 -19894.473,E2 -19894.473} C_VEL
LIN {X 0,Y 225.809,Z 396.434,A -85,B 0,C 180,E1 -19897.152,E2 -19897.152} C_VEL
LIN {X 0,Y 226.337,Z 393.488,A -85,B 0,C 180,E1 -19899.833,E2 -19899.833} C_VEL
LIN {X 0,Y 227.25,Z 389.506,A -85,B 0,C 180,E1 -19902.503,E2 -19902.503} C_VEL
LIN {X 0,Y 228.859,Z 383.385,A -85,B 0,C 180,E1 -19905.587,E2 -19905.587} C_VEL
LIN {X 0,Y 230.692,Z 376.703,A -85,B 0,C 180,E1 -19908.196,E2 -19908.196} C_VEL
LIN {X 0,Y 232.649,Z 369.242,A -85,B 0,C 180,E1 -19910.533,E2 -19910.533} C_VEL
LIN {X 0,Y 235.093,Z 359.914,A -85,B 0,C 180,E1 -19912.869,E2 -19912.869} C_VEL
LIN {X 0,Y 237.704,Z 349.415,A -85,B 0,C 180,E1 -19914.918,E2 -19914.918} C_VEL
LIN {X 0,Y 240.303,Z 337.596,A -85,B 0,C 180,E1 -19916.722,E2 -19916.722} C_VEL
LIN {X 0,Y 242.455,Z 325.683,A -85,B 0,C 180,E1 -19918.101,E2 -19918.101} C_VEL
LIN {X 0,Y 244.33,Z 313.283,A -85,B 0,C 180,E1 -19919.156,E2 -19919.156} C_VEL
LIN {X 0,Y 245.797,Z 300.636,A -85,B 0,C 180,E1 -19919.898,E2 -19919.898} C_VEL
LIN {X 0,Y 246.578,Z 287.363,A -85,B 0,C 180,E1 -19920.378,E2 -19920.378} C_VEL
LIN {X 0,Y 248.267,Z 238.303,A -85,B 0,C 180,E1 -19921.769,E2 -19921.769} C_VEL
LIN {X 0,Y 245.541,Z 220.648,A -85,B 0,C 180,E1 -19922.759,E2 -19922.759} C_VEL
LIN {X 0,Y 238.715,Z 204.335,A -85,B 0,C 180,E1 -19924.392,E2 -19924.392} C_VEL
LIN {X 0,Y 232.344,Z 191.024,A -85,B 0,C 180,E1 -19925.962,E2 -19925.962} C_VEL
LIN {X 0,Y 230.255,Z 186.793,A -85,B 0,C 180,E1 -19926.535,E2 -19926.535} C_VEL
LIN {X 0,Y 228.002,Z 178.475,A -85,B 0,C 180,E1 -19930.679,E2 -19930.679} C_VEL
LIN {X 0,Y 227.821,Z 177.609,A -85,B 0,C 180,E1 -19931.15,E2 -19931.15} C_VEL
LIN {X 0,Y 227.825,Z 177.608,A -85,B 0,C 180,E1 -19935.195,E2 -19935.195} C_VEL
LIN {X 0,Y 227.825,Z 177.606,A -85,B 0,C 180,E1 -19939.623,E2 -19939.623} C_VEL
LIN {X 0,Y 227.881,Z 177.599,A -85,B 0,C 180,E1 -19944.128,E2 -19944.128} C_VEL
LIN {X 0,Y 227.856,Z 177.604,A -85,B 0,C 180,E1 -19948.376,E2 -19948.376} C_VEL
LIN {X 0,Y 227.856,Z 177.596,A -85,B 0,C 180,E1 -19952.441,E2 -19952.441} C_VEL
LIN {X 0,Y 227.899,Z 177.592,A -85,B 0,C 180,E1 -19956.366,E2 -19956.366} C_VEL
LIN {X 0,Y 227.937,Z 177.591,A -85,B 0,C 180,E1 -19960.174,E2 -19960.174} C_VEL
LIN {X 0,Y 228.058,Z 177.576,A -85,B 0,C 180,E1 -19963.898,E2 -19963.898} C_VEL
LIN {X 0,Y 228.073,Z 177.567,A -85,B 0,C 180,E1 -19967.543,E2 -19967.543} C_VEL
LIN {X 0,Y 228.268,Z 177.552,A -85,B 0,C 180,E1 -19971.145,E2 -19971.145} C_VEL
LIN {X 0,Y 228.324,Z 177.536,A -85,B 0,C 180,E1 -19972.928,E2 -19972.928} C_VEL
LIN {X 0,Y 228.555,Z 177.51,A -85,B 0,C 180,E1 -19978.238,E2 -19978.238} C_VEL
LIN {X 0,Y 228.554,Z 177.515,A -85,B 0,C 180,E1 -19981.762,E2 -19981.762} C_VEL
LIN {X 0,Y 228.324,Z 177.539,A -85,B 0,C 180,E1 -19987.073,E2 -19987.073} C_VEL
LIN {X 0,Y 228.146,Z 177.559,A -85,B 0,C 180,E1 -19990.651,E2 -19990.651} C_VEL
LIN {X 0,Y 228.066,Z 177.576,A -85,B 0,C 180,E1 -19994.272,E2 -19994.272} C_VEL
LIN {X 0,Y 228.004,Z 177.576,A -85,B 0,C 180,E1 -19997.953,E2 -19997.953} C_VEL
LIN {X 0,Y 227.931,Z 177.586,A -85,B 0,C 180,E1 -20002.329,E2 -20002.329} C_VEL
LIN {X 0,Y 227.944,Z 177.586,A -85,B 0,C 180,E1 -20006.603,E2 -20006.603} C_VEL
LIN {X 0,Y 227.91,Z 177.596,A -85,B 0,C 180,E1 -20010.296,E2 -20010.296} C_VEL
LIN {X 0,Y 227.891,Z 177.597,A -85,B 0,C 180,E1 -20013.718,E2 -20013.718} C_VEL
LIN {X 0,Y 227.871,Z 177.601,A -85,B 0,C 180,E1 -20018.086,E2 -20018.086} C_VEL
LIN {X 0,Y 227.814,Z 177.604,A -85,B 0,C 180,E1 -20022.742,E2 -20022.742} C_VEL
LIN {X 0,Y 227.812,Z 177.606,A -85,B 0,C 180,E1 -20027.258,E2 -20027.258} C_VEL
LIN {X 0,Y 227.846,Z 177.603,A -85,B 0,C 180,E1 -20031.909,E2 -20031.909} C_VEL
LIN {X 0,Y 227.889,Z 177.738,A -85,B 0,C 180,E1 -20032.689,E2 -20032.689} C_VEL
LIN {X 0,Y 228.081,Z 178.612,A -85,B 0,C 180,E1 -20033.142,E2 -20033.142} C_VEL
LIN {X 0,Y 230.196,Z 182.503,A -85,B 0,C 180,E1 -20033.695,E2 -20033.695} C_VEL
LIN {X 0,Y 237.242,Z 195.77,A -85,B 0,C 180,E1 -20035.424,E2 -20035.424} C_VEL
LIN {X 0,Y 243.854,Z 209.805,A -85,B 0,C 180,E1 -20036.981,E2 -20036.981} C_VEL
LIN {X 0,Y 248.915,Z 222.439,A -85,B 0,C 180,E1 -20038.162,E2 -20038.162} C_VEL
LIN {X 0,Y 246.638,Z 283.324,A -85,B 0,C 180,E1 -20039.886,E2 -20039.886} C_VEL
LIN {X 0,Y 245.688,Z 296.08,A -85,B 0,C 180,E1 -20040.468,E2 -20040.468} C_VEL
LIN {X 0,Y 244.115,Z 309.184,A -85,B 0,C 180,E1 -20041.404,E2 -20041.404} C_VEL
LIN {X 0,Y 242.319,Z 321.02,A -85,B 0,C 180,E1 -20042.586,E2 -20042.586} C_VEL
LIN {X 0,Y 240.23,Z 331.766,A -85,B 0,C 180,E1 -20043.971,E2 -20043.971} C_VEL
LIN {X 0,Y 237.824,Z 342.716,A -85,B 0,C 180,E1 -20045.794,E2 -20045.794} C_VEL
LIN {X 0,Y 235.63,Z 352.17,A -85,B 0,C 180,E1 -20047.794,E2 -20047.794} C_VEL
LIN {X 0,Y 233.694,Z 359.771,A -85,B 0,C 180,E1 -20049.767,E2 -20049.767} C_VEL
LIN {X 0,Y 231.326,Z 367.773,A -85,B 0,C 180,E1 -20052.313,E2 -20052.313} C_VEL
LIN {X 0,Y 229.532,Z 374.189,A -85,B 0,C 180,E1 -20054.915,E2 -20054.915} C_VEL
LIN {X 0,Y 228.032,Z 379.279,A -85,B 0,C 180,E1 -20057.541,E2 -20057.541} C_VEL
LIN {X 0,Y 226.986,Z 383.229,A -85,B 0,C 180,E1 -20060.195,E2 -20060.195} C_VEL
LIN {X 0,Y 226.321,Z 386.145,A -85,B 0,C 180,E1 -20062.865,E2 -20062.865} C_VEL
LIN {X 0,Y 225.992,Z 387.54,A -85,B 0,C 180,E1 -20064.647,E2 -20064.647} C_VEL
LIN {X 0,Y 225.819,Z 388.531,A -85,B 0,C 180,E1 -20066.431,E2 -20066.431} C_VEL
LIN {X 0,Y 225.722,Z 389.141,A -85,B 0,C 180,E1 -20068.216,E2 -20068.216} C_VEL
LIN {X 0,Y 225.684,Z 389.37,A -85,B 0,C 180,E1 -20070,E2 -20070} C_VEL
LIN {X 0,Y 225.722,Z 389.176,A -85,B 0,C 180,E1 -20071.784,E2 -20071.784} C_VEL
LIN {X 0,Y 225.811,Z 388.59,A -85,B 0,C 180,E1 -20073.569,E2 -20073.569} C_VEL
LIN {X 0,Y 226.036,Z 387.369,A -85,B 0,C 180,E1 -20075.754,E2 -20075.754} C_VEL
LIN {X 0,Y 226.691,Z 384.449,A -85,B 0,C 180,E1 -20078.917,E2 -20078.917} C_VEL
LIN {X 0,Y 227.597,Z 380.913,A -85,B 0,C 180,E1 -20081.579,E2 -20081.579} C_VEL
LIN {X 0,Y 228.922,Z 376.272,A -85,B 0,C 180,E1 -20084.217,E2 -20084.217} C_VEL
LIN {X 0,Y 230.906,Z 369.277,A -85,B 0,C 180,E1 -20087.263,E2 -20087.263} C_VEL
LIN {X 0,Y 233.22,Z 361.689,A -85,B 0,C 180,E1 -20089.817,E2 -20089.817} C_VEL
LIN {X 0,Y 235.295,Z 353.605,A -85,B 0,C 180,E1 -20092.005,E2 -20092.005} C_VEL
LIN {X 0,Y 237.773,Z 343.357,A -85,B 0,C 180,E1 -20094.212,E2 -20094.212} C_VEL
LIN {X 0,Y 240.196,Z 332.587,A -85,B 0,C 180,E1 -20096.033,E2 -20096.033} C_VEL
LIN {X 0,Y 242.219,Z 322.074,A -85,B 0,C 180,E1 -20097.427,E2 -20097.427} C_VEL
LIN {X 0,Y 244.255,Z 309.412,A -85,B 0,C 180,E1 -20098.695,E2 -20098.695} C_VEL
LIN {X 0,Y 245.635,Z 296.774,A -85,B 0,C 180,E1 -20099.629,E2 -20099.629} C_VEL
LIN {X 0,Y 246.713,Z 284.781,A -85,B 0,C 180,E1 -20100.187,E2 -20100.187} C_VEL
LIN {X 0,Y 249.064,Z 222.868,A -85,B 0,C 180,E1 -20101.944,E2 -20101.944} C_VEL
LIN {X 0,Y 243.948,Z 209.912,A -85,B 0,C 180,E1 -20103.146,E2 -20103.146} C_VEL
LIN {X 0,Y 236.338,Z 193.851,A -85,B 0,C 180,E1 -20104.948,E2 -20104.948} C_VEL
LIN {X 0,Y 229.951,Z 182.147,A -85,B 0,C 180,E1 -20106.519,E2 -20106.519} C_VEL
LIN {X 0,Y 228.114,Z 178.599,A -85,B 0,C 180,E1 -20107.016,E2 -20107.016} C_VEL
LIN {X 0,Y 227.86,Z 177.599,A -85,B 0,C 180,E1 -20107.612,E2 -20107.612} C_VEL
LIN {X 0,Y 227.812,Z 177.605,A -85,B 0,C 180,E1 -20112.234,E2 -20112.234} C_VEL
LIN {X 0,Y 227.834,Z 177.601,A -85,B 0,C 180,E1 -20115.192,E2 -20115.192} C_VEL
LIN {X 0,Y 227.834,Z 177.603,A -85,B 0,C 180,E1 -20119.625,E2 -20119.625} C_VEL
LIN {X 0,Y 227.9,Z 177.597,A -85,B 0,C 180,E1 -20124.131,E2 -20124.131} C_VEL
LIN {X 0,Y 227.872,Z 177.599,A -85,B 0,C 180,E1 -20128.378,E2 -20128.378} C_VEL
LIN {X 0,Y 227.886,Z 177.589,A -85,B 0,C 180,E1 -20132.445,E2 -20132.445} C_VEL
LIN {X 0,Y 227.914,Z 177.59,A -85,B 0,C 180,E1 -20136.367,E2 -20136.367} C_VEL
LIN {X 0,Y 227.943,Z 177.59,A -85,B 0,C 180,E1 -20140.174,E2 -20140.174} C_VEL
LIN {X 0,Y 228.058,Z 177.563,A -85,B 0,C 180,E1 -20143.898,E2 -20143.898} C_VEL
LIN {X 0,Y 228.094,Z 177.573,A -85,B 0,C 180,E1 -20147.544,E2 -20147.544} C_VEL
LIN {X 0,Y 228.305,Z 177.532,A -85,B 0,C 180,E1 -20151.146,E2 -20151.146} C_VEL
LIN {X 0,Y 228.353,Z 177.531,A -85,B 0,C 180,E1 -20152.928,E2 -20152.928} C_VEL
LIN {X 0,Y 228.554,Z 177.502,A -85,B 0,C 180,E1 -20158.238,E2 -20158.238} C_VEL
LIN {X 0,Y 228.554,Z 177.514,A -85,B 0,C 180,E1 -20161.762,E2 -20161.762} C_VEL
LIN {X 0,Y 228.353,Z 177.529,A -85,B 0,C 180,E1 -20167.071,E2 -20167.071} C_VEL
LIN {X 0,Y 228.159,Z 177.562,A -85,B 0,C 180,E1 -20170.651,E2 -20170.651} C_VEL
LIN {X 0,Y 228.064,Z 177.565,A -85,B 0,C 180,E1 -20174.272,E2 -20174.272} C_VEL
LIN {X 0,Y 228.002,Z 177.578,A -85,B 0,C 180,E1 -20177.953,E2 -20177.953} C_VEL
LIN {X 0,Y 227.917,Z 177.595,A -85,B 0,C 180,E1 -20182.321,E2 -20182.321} C_VEL
LIN {X 0,Y 227.941,Z 177.589,A -85,B 0,C 180,E1 -20186.602,E2 -20186.602} C_VEL
LIN {X 0,Y 227.857,Z 177.597,A -85,B 0,C 180,E1 -20188.148,E2 -20188.148} C_VEL
LIN {X 0,Y 227.174,Z 177.683,A -85,B 0,C 180,E1 -20189.623,E2 -20189.623} C_VEL
LIN {X 0,Y 224.303,Z 178.046,A -85,B 0,C 180,E1 -20192.031,E2 -20192.031} C_VEL
LIN {X 0,Y 221.877,Z 178.342,A -85,B 0,C 180,E1 -20193.995,E2 -20193.995} C_VEL
LIN {X 0,Y 220.848,Z 178.471,A -85,B 0,C 180,E1 -20195.521,E2 -20195.521} C_VEL
LIN {X 0,Y 220.77,Z 178.475,A -85,B 0,C 180,E1 -20196.038,E2 -20196.038} C_VEL
LIN {X 0,Y 220.794,Z 178.482,A -85,B 0,C 180,E1 -20200.188,E2 -20200.188} C_VEL
LIN {X 0,Y 220.766,Z 178.481,A -85,B 0,C 180,E1 -20204.456,E2 -20204.456} C_VEL
LIN {X 0,Y 220.783,Z 178.63,A -85,B 0,C 180,E1 -20207.796,E2 -20207.796} C_VEL
LIN {X 0,Y 223.013,Z 186.773,A -85,B 0,C 180,E1 -20212.052,E2 -20212.052} C_VEL
LIN {X 0,Y 225.052,Z 190.794,A -85,B 0,C 180,E1 -20212.611,E2 -20212.611} C_VEL
LIN {X 0,Y 231.585,Z 203.701,A -85,B 0,C 180,E1 -20214.314,E2 -20214.314} C_VEL
LIN {X 0,Y 238.66,Z 220.18,A -85,B 0,C 180,E1 -20216.105,E2 -20216.105} C_VEL
LIN {X 0,Y 240.195,Z 224.512,A -85,B 0,C 180,E1 -20216.501,E2 -20216.501} C_VEL
LIN {X 0,Y 242.378,Z 240.175,A -85,B 0,C 180,E1 -20217.381,E2 -20217.381} C_VEL
LIN {X 0,Y 240.083,Z 296.059,A -85,B 0,C 180,E1 -20219.022,E2 -20219.022} C_VEL
LIN {X 0,Y 238.714,Z 309.601,A -85,B 0,C 180,E1 -20219.728,E2 -20219.728} C_VEL
LIN {X 0,Y 236.955,Z 321.966,A -85,B 0,C 180,E1 -20220.7,E2 -20220.7} C_VEL
LIN {X 0,Y 234.683,Z 334.636,A -85,B 0,C 180,E1 -20222.101,E2 -20222.101} C_VEL
LIN {X 0,Y 232.178,Z 345.904,A -85,B 0,C 180,E1 -20223.724,E2 -20223.724} C_VEL
LIN {X 0,Y 229.6,Z 356.053,A -85,B 0,C 180,E1 -20225.592,E2 -20225.592} C_VEL
LIN {X 0,Y 227.132,Z 365.2,A -85,B 0,C 180,E1 -20227.726,E2 -20227.726} C_VEL
LIN {X 0,Y 225.147,Z 372.762,A -85,B 0,C 180,E1 -20229.918,E2 -20229.918} C_VEL
LIN {X 0,Y 222.973,Z 380.181,A -85,B 0,C 180,E1 -20232.577,E2 -20232.577} C_VEL
LIN {X 0,Y 221.112,Z 386.138,A -85,B 0,C 180,E1 -20235.269,E2 -20235.269} C_VEL
LIN {X 0,Y 219.908,Z 390.851,A -85,B 0,C 180,E1 -20238.011,E2 -20238.011} C_VEL
LIN {X 0,Y 219.09,Z 394.452,A -85,B 0,C 180,E1 -20240.771,E2 -20240.771} C_VEL
LIN {X 0,Y 218.736,Z 396.309,A -85,B 0,C 180,E1 -20242.616,E2 -20242.616} C_VEL
LIN {X 0,Y 218.498,Z 398.699,A -85,B 0,C 180,E1 -20246.312,E2 -20246.312} C_VEL
LIN {X 0,Y 218.517,Z 399.307,A -85,B 0,C 180,E1 -20248.157,E2 -20248.157} C_VEL
LIN {X 0,Y 218.59,Z 399.52,A -85,B 0,C 180,E1 -20250,E2 -20250} C_VEL
LIN {X 0,Y 218.518,Z 399.295,A -85,B 0,C 180,E1 -20251.843,E2 -20251.843} C_VEL
LIN {X 0,Y 218.481,Z 398.415,A -85,B 0,C 180,E1 -20254.292,E2 -20254.292} C_VEL
LIN {X 0,Y 218.736,Z 396.271,A -85,B 0,C 180,E1 -20257.384,E2 -20257.384} C_VEL
LIN {X 0,Y 219.323,Z 393.325,A -85,B 0,C 180,E1 -20260.151,E2 -20260.151} C_VEL
LIN {X 0,Y 220.27,Z 389.341,A -85,B 0,C 180,E1 -20262.906,E2 -20262.906} C_VEL
LIN {X 0,Y 222.01,Z 383.221,A -85,B 0,C 180,E1 -20266.081,E2 -20266.081} C_VEL
LIN {X 0,Y 223.93,Z 376.538,A -85,B 0,C 180,E1 -20268.765,E2 -20268.765} C_VEL
LIN {X 0,Y 226.022,Z 368.887,A -85,B 0,C 180,E1 -20271.225,E2 -20271.225} C_VEL
LIN {X 0,Y 228.548,Z 359.748,A -85,B 0,C 180,E1 -20273.563,E2 -20273.563} C_VEL
LIN {X 0,Y 231.256,Z 349.249,A -85,B 0,C 180,E1 -20275.662,E2 -20275.662} C_VEL
LIN {X 0,Y 233.979,Z 337.429,A -85,B 0,C 180,E1 -20277.504,E2 -20277.504} C_VEL
LIN {X 0,Y 236.21,Z 325.514,A -85,B 0,C 180,E1 -20278.913,E2 -20278.913} C_VEL
LIN {X 0,Y 238.162,Z 313.113,A -85,B 0,C 180,E1 -20279.988,E2 -20279.988} C_VEL
LIN {X 0,Y 239.729,Z 299.933,A -85,B 0,C 180,E1 -20280.767,E2 -20280.767} C_VEL
LIN {X 0,Y 240.593,Z 285.103,A -85,B 0,C 180,E1 -20281.288,E2 -20281.288} C_VEL
LIN {X 0,Y 242.238,Z 239.488,A -85,B 0,C 180,E1 -20282.609,E2 -20282.609} C_VEL
LIN {X 0,Y 239.819,Z 223.348,A -85,B 0,C 180,E1 -20283.542,E2 -20283.542} C_VEL
LIN {X 0,Y 233.446,Z 207.955,A -85,B 0,C 180,E1 -20285.142,E2 -20285.142} C_VEL
LIN {X 0,Y 227.274,Z 195.035,A -85,B 0,C 180,E1 -20286.734,E2 -20286.734} C_VEL
LIN {X 0,Y 222.938,Z 186.617,A -85,B 0,C 180,E1 -20287.925,E2 -20287.925} C_VEL
LIN {X 0,Y 220.765,Z 178.487,A -85,B 0,C 180,E1 -20292.255,E2 -20292.255} C_VEL
LIN {X 0,Y 220.761,Z 178.486,A -85,B 0,C 180,E1 -20297.072,E2 -20297.072} C_VEL
LIN {X 0,Y 220.806,Z 178.481,A -85,B 0,C 180,E1 -20300.463,E2 -20300.463} C_VEL
LIN {X 0,Y 220.801,Z 178.481,A -85,B 0,C 180,E1 -20305.045,E2 -20305.045} C_VEL
LIN {X 0,Y 220.834,Z 178.477,A -85,B 0,C 180,E1 -20309.39,E2 -20309.39} C_VEL
LIN {X 0,Y 220.876,Z 178.466,A -85,B 0,C 180,E1 -20313.547,E2 -20313.547} C_VEL
LIN {X 0,Y 220.87,Z 178.465,A -85,B 0,C 180,E1 -20317.553,E2 -20317.553} C_VEL
LIN {X 0,Y 220.985,Z 178.45,A -85,B 0,C 180,E1 -20322.571,E2 -20322.571} C_VEL
LIN {X 0,Y 221.012,Z 178.447,A -85,B 0,C 180,E1 -20327.139,E2 -20327.139} C_VEL
LIN {X 0,Y 221.205,Z 178.43,A -85,B 0,C 180,E1 -20330.859,E2 -20330.859} C_VEL
LIN {X 0,Y 221.26,Z 178.417,A -85,B 0,C 180,E1 -20332.701,E2 -20332.701} C_VEL
LIN {X 0,Y 221.513,Z 178.387,A -85,B 0,C 180,E1 -20338.182,E2 -20338.182} C_VEL
LIN {X 0,Y 221.512,Z 178.392,A -85,B 0,C 180,E1 -20341.818,E2 -20341.818} C_VEL
LIN {X 0,Y 221.259,Z 178.421,A -85,B 0,C 180,E1 -20347.3,E2 -20347.3} C_VEL
LIN {X 0,Y 221.068,Z 178.438,A -85,B 0,C 180,E1 -20350.996,E2 -20350.996} C_VEL
LIN {X 0,Y 220.997,Z 178.458,A -85,B 0,C 180,E1 -20354.739,E2 -20354.739} C_VEL
LIN {X 0,Y 220.923,Z 178.46,A -85,B 0,C 180,E1 -20358.549,E2 -20358.549} C_VEL
LIN {X 0,Y 220.897,Z 178.461,A -85,B 0,C 180,E1 -20362.683,E2 -20362.683} C_VEL
LIN {X 0,Y 220.887,Z 178.463,A -85,B 0,C 180,E1 -20367.016,E2 -20367.016} C_VEL
LIN {X 0,Y 220.864,Z 178.47,A -85,B 0,C 180,E1 -20370.779,E2 -20370.779} C_VEL
LIN {X 0,Y 220.816,Z 178.477,A -85,B 0,C 180,E1 -20374.953,E2 -20374.953} C_VEL
LIN {X 0,Y 220.839,Z 178.476,A -85,B 0,C 180,E1 -20377.288,E2 -20377.288} C_VEL
LIN {X 0,Y 220.775,Z 178.481,A -85,B 0,C 180,E1 -20381.952,E2 -20381.952} C_VEL
LIN {X 0,Y 220.775,Z 178.48,A -85,B 0,C 180,E1 -20385.546,E2 -20385.546} C_VEL
LIN {X 0,Y 220.808,Z 178.478,A -85,B 0,C 180,E1 -20390.463,E2 -20390.463} C_VEL
LIN {X 0,Y 220.827,Z 178.675,A -85,B 0,C 180,E1 -20391.646,E2 -20391.646} C_VEL
LIN {X 0,Y 222.023,Z 181.662,A -85,B 0,C 180,E1 -20392.085,E2 -20392.085} C_VEL
LIN {X 0,Y 223.668,Z 183.92,A -85,B 0,C 180,E1 -20392.504,E2 -20392.504} C_VEL
LIN {X 0,Y 230.165,Z 195.693,A -85,B 0,C 180,E1 -20394.189,E2 -20394.189} C_VEL
LIN {X 0,Y 237.713,Z 211.538,A -85,B 0,C 180,E1 -20396.068,E2 -20396.068} C_VEL
LIN {X 0,Y 242.859,Z 224.347,A -85,B 0,C 180,E1 -20397.33,E2 -20397.33} C_VEL
LIN {X 0,Y 240.561,Z 283.193,A -85,B 0,C 180,E1 -20399.031,E2 -20399.031} C_VEL
LIN {X 0,Y 239.532,Z 296.468,A -85,B 0,C 180,E1 -20399.646,E2 -20399.646} C_VEL
LIN {X 0,Y 237.92,Z 309.354,A -85,B 0,C 180,E1 -20400.588,E2 -20400.588} C_VEL
LIN {X 0,Y 236.05,Z 321.188,A -85,B 0,C 180,E1 -20401.793,E2 -20401.793} C_VEL
LIN {X 0,Y 233.88,Z 331.932,A -85,B 0,C 180,E1 -20403.209,E2 -20403.209} C_VEL
LIN {X 0,Y 231.361,Z 342.882,A -85,B 0,C 180,E1 -20405.072,E2 -20405.072} C_VEL
LIN {X 0,Y 228.899,Z 352.959,A -85,B 0,C 180,E1 -20407.273,E2 -20407.273} C_VEL
LIN {X 0,Y 226.612,Z 361.416,A -85,B 0,C 180,E1 -20409.58,E2 -20409.58} C_VEL
LIN {X 0,Y 224.195,Z 369.106,A -85,B 0,C 180,E1 -20412.203,E2 -20412.203} C_VEL
LIN {X 0,Y 222.097,Z 376.162,A -85,B 0,C 180,E1 -20415.336,E2 -20415.336} C_VEL
LIN {X 0,Y 220.654,Z 380.861,A -85,B 0,C 180,E1 -20418.052,E2 -20418.052} C_VEL
LIN {X 0,Y 219.701,Z 384.453,A -85,B 0,C 180,E1 -20420.796,E2 -20420.796} C_VEL
LIN {X 0,Y 219.272,Z 386.308,A -85,B 0,C 180,E1 -20422.634,E2 -20422.634} C_VEL
LIN {X 0,Y 218.927,Z 387.702,A -85,B 0,C 180,E1 -20424.473,E2 -20424.473} C_VEL
LIN {X 0,Y 218.643,Z 389.303,A -85,B 0,C 180,E1 -20428.158,E2 -20428.158} C_VEL
LIN {X 0,Y 218.602,Z 389.532,A -85,B 0,C 180,E1 -20430,E2 -20430} C_VEL
LIN {X 0,Y 218.642,Z 389.338,A -85,B 0,C 180,E1 -20431.842,E2 -20431.842} C_VEL
LIN {X 0,Y 218.907,Z 387.784,A -85,B 0,C 180,E1 -20435.527,E2 -20435.527} C_VEL
LIN {X 0,Y 219.208,Z 386.425,A -85,B 0,C 180,E1 -20437.368,E2 -20437.368} C_VEL
LIN {X 0,Y 219.936,Z 383.554,A -85,B 0,C 180,E1 -20440.122,E2 -20440.122} C_VEL
LIN {X 0,Y 221.05,Z 379.659,A -85,B 0,C 180,E1 -20442.859,E2 -20442.859} C_VEL
LIN {X 0,Y 222.599,Z 374.633,A -85,B 0,C 180,E1 -20445.567,E2 -20445.567} C_VEL
LIN {X 0,Y 224.538,Z 368.302,A -85,B 0,C 180,E1 -20448.24,E2 -20448.24} C_VEL
LIN {X 0,Y 226.984,Z 360.378,A -85,B 0,C 180,E1 -20450.859,E2 -20450.859} C_VEL
LIN {X 0,Y 229.022,Z 352.486,A -85,B 0,C 180,E1 -20452.984,E2 -20452.984} C_VEL
LIN {X 0,Y 231.583,Z 342.449,A -85,B 0,C 180,E1 -20455.142,E2 -20455.142} C_VEL
LIN {X 0,Y 233.859,Z 332.744,A -85,B 0,C 180,E1 -20456.794,E2 -20456.794} C_VEL
LIN {X 0,Y 235.955,Z 322.23,A -85,B 0,C 180,E1 -20458.219,E2 -20458.219} C_VEL
LIN {X 0,Y 238.064,Z 309.566,A -85,B 0,C 180,E1 -20459.514,E2 -20459.514} C_VEL
LIN {X 0,Y 239.481,Z 297.15,A -85,B 0,C 180,E1 -20460.452,E2 -20460.452} C_VEL
LIN {X 0,Y 240.624,Z 284.525,A -85,B 0,C 180,E1 -20461.05,E2 -20461.05} C_VEL
LIN {X 0,Y 243.003,Z 224.581,A -85,B 0,C 180,E1 -20462.785,E2 -20462.785} C_VEL
LIN {X 0,Y 238.355,Z 212.965,A -85,B 0,C 180,E1 -20463.924,E2 -20463.924} C_VEL
LIN {X 0,Y 232.155,Z 199.69,A -85,B 0,C 180,E1 -20465.459,E2 -20465.459} C_VEL
LIN {X 0,Y 225.483,Z 186.978,A -85,B 0,C 180,E1 -20467.179,E2 -20467.179} C_VEL
LIN {X 0,Y 222.692,Z 182.459,A -85,B 0,C 180,E1 -20467.909,E2 -20467.909} C_VEL
LIN {X 0,Y 221.176,Z 179.994,A -85,B 0,C 180,E1 -20468.317,E2 -20468.317} C_VEL
LIN {X 0,Y 220.827,Z 178.703,A -85,B 0,C 180,E1 -20468.505,E2 -20468.505} C_VEL
LIN {X 0,Y 220.808,Z 178.477,A -85,B 0,C 180,E1 -20469.536,E2 -20469.536} C_VEL
LIN {X 0,Y 220.774,Z 178.48,A -85,B 0,C 180,E1 -20474.454,E2 -20474.454} C_VEL
LIN {X 0,Y 220.775,Z 178.478,A -85,B 0,C 180,E1 -20478.048,E2 -20478.048} C_VEL
LIN {X 0,Y 220.831,Z 178.47,A -85,B 0,C 180,E1 -20482.794,E2 -20482.794} C_VEL
LIN {X 0,Y 220.823,Z 178.467,A -85,B 0,C 180,E1 -20487.245,E2 -20487.245} C_VEL
LIN {X 0,Y 220.837,Z 178.466,A -85,B 0,C 180,E1 -20491.486,E2 -20491.486} C_VEL
LIN {X 0,Y 220.868,Z 178.472,A -85,B 0,C 180,E1 -20495.565,E2 -20495.565} C_VEL
LIN {X 0,Y 220.893,Z 178.464,A -85,B 0,C 180,E1 -20499.514,E2 -20499.514} C_VEL
LIN {X 0,Y 221.017,Z 178.442,A -85,B 0,C 180,E1 -20503.37,E2 -20503.37} C_VEL
LIN {X 0,Y 221.112,Z 178.44,A -85,B 0,C 180,E1 -20509.006,E2 -20509.006} C_VEL
LIN {X 0,Y 221.289,Z 178.409,A -85,B 0,C 180,E1 -20512.701,E2 -20512.701} C_VEL
LIN {X 0,Y 221.512,Z 178.378,A -85,B 0,C 180,E1 -20518.182,E2 -20518.182} C_VEL
LIN {X 0,Y 221.512,Z 178.391,A -85,B 0,C 180,E1 -20521.818,E2 -20521.818} C_VEL
LIN {X 0,Y 221.289,Z 178.41,A -85,B 0,C 180,E1 -20527.298,E2 -20527.298} C_VEL
LIN {X 0,Y 221.107,Z 178.438,A -85,B 0,C 180,E1 -20530.994,E2 -20530.994} C_VEL
LIN {X 0,Y 221.016,Z 178.453,A -85,B 0,C 180,E1 -20536.63,E2 -20536.63} C_VEL
LIN {X 0,Y 220.884,Z 178.46,A -85,B 0,C 180,E1 -20540.487,E2 -20540.487} C_VEL
LIN {X 0,Y 220.862,Z 178.464,A -85,B 0,C 180,E1 -20544.436,E2 -20544.436} C_VEL
LIN {X 0,Y 220.827,Z 178.476,A -85,B 0,C 180,E1 -20548.515,E2 -20548.515} C_VEL
LIN {X 0,Y 220.816,Z 178.479,A -85,B 0,C 180,E1 -20552.756,E2 -20552.756} C_VEL
LIN {X 0,Y 220.77,Z 178.475,A -85,B 0,C 180,E1 -20556.038,E2 -20556.038} C_VEL
LIN {X 0,Y 220.123,Z 178.564,A -85,B 0,C 180,E1 -20557.561,E2 -20557.561} C_VEL
LIN {X 0,Y 217.296,Z 178.92,A -85,B 0,C 180,E1 -20560.047,E2 -20560.047} C_VEL
LIN {X 0,Y 214.023,Z 179.327,A -85,B 0,C 180,E1 -20563.122,E2 -20563.122} C_VEL
LIN {X 0,Y 213.667,Z 179.363,A -85,B 0,C 180,E1 -20564.187,E2 -20564.187} C_VEL
LIN {X 0,Y 213.73,Z 179.456,A -85,B 0,C 180,E1 -20566.594,E2 -20566.594} C_VEL
LIN {X 0,Y 215.686,Z 186.626,A -85,B 0,C 180,E1 -20570.519,E2 -20570.519} C_VEL
LIN {X 0,Y 217.945,Z 190.801,A -85,B 0,C 180,E1 -20571.177,E2 -20571.177} C_VEL
LIN {X 0,Y 224.847,Z 204.113,A -85,B 0,C 180,E1 -20573.094,E2 -20573.094} C_VEL
LIN {X 0,Y 231.62,Z 219.323,A -85,B 0,C 180,E1 -20574.901,E2 -20574.901} C_VEL
LIN {X 0,Y 234.475,Z 227.001,A -85,B 0,C 180,E1 -20575.666,E2 -20575.666} C_VEL
LIN {X 0,Y 236.407,Z 241.285,A -85,B 0,C 180,E1 -20576.494,E2 -20576.494} C_VEL
LIN {X 0,Y 234.048,Z 295.594,A -85,B 0,C 180,E1 -20578.113,E2 -20578.113} C_VEL
LIN {X 0,Y 232.727,Z 308.834,A -85,B 0,C 180,E1 -20578.813,E2 -20578.813} C_VEL
LIN {X 0,Y 230.964,Z 320.703,A -85,B 0,C 180,E1 -20579.737,E2 -20579.737} C_VEL
LIN {X 0,Y 228.779,Z 332.896,A -85,B 0,C 180,E1 -20581.064,E2 -20581.064} C_VEL
LIN {X 0,Y 226.149,Z 344.452,A -85,B 0,C 180,E1 -20582.717,E2 -20582.717} C_VEL
LIN {X 0,Y 223.435,Z 354.859,A -85,B 0,C 180,E1 -20584.624,E2 -20584.624} C_VEL
LIN {X 0,Y 221.042,Z 363.37,A -85,B 0,C 180,E1 -20586.582,E2 -20586.582} C_VEL
LIN {X 0,Y 218.954,Z 371.051,A -85,B 0,C 180,E1 -20588.772,E2 -20588.772} C_VEL
LIN {X 0,Y 216.475,Z 378.899,A -85,B 0,C 180,E1 -20591.546,E2 -20591.546} C_VEL
LIN {X 0,Y 214.239,Z 385.977,A -85,B 0,C 180,E1 -20594.786,E2 -20594.786} C_VEL
LIN {X 0,Y 212.932,Z 390.689,A -85,B 0,C 180,E1 -20597.612,E2 -20597.612} C_VEL
LIN {X 0,Y 212.064,Z 394.29,A -85,B 0,C 180,E1 -20600.462,E2 -20600.462} C_VEL
LIN {X 0,Y 211.67,Z 396.147,A -85,B 0,C 180,E1 -20602.368,E2 -20602.368} C_VEL
LIN {X 0,Y 211.397,Z 398.537,A -85,B 0,C 180,E1 -20606.188,E2 -20606.188} C_VEL
LIN {X 0,Y 211.42,Z 399.145,A -85,B 0,C 180,E1 -20608.095,E2 -20608.095} C_VEL
LIN {X 0,Y 211.49,Z 399.358,A -85,B 0,C 180,E1 -20610,E2 -20610} C_VEL
LIN {X 0,Y 211.42,Z 399.133,A -85,B 0,C 180,E1 -20611.905,E2 -20611.905} C_VEL
LIN {X 0,Y 211.393,Z 398.376,A -85,B 0,C 180,E1 -20614.145,E2 -20614.145} C_VEL
LIN {X 0,Y 211.67,Z 396.107,A -85,B 0,C 180,E1 -20617.632,E2 -20617.632} C_VEL
LIN {X 0,Y 212.328,Z 393.161,A -85,B 0,C 180,E1 -20620.489,E2 -20620.489} C_VEL
LIN {X 0,Y 213.304,Z 389.176,A -85,B 0,C 180,E1 -20623.335,E2 -20623.335} C_VEL
LIN {X 0,Y 215.154,Z 383.056,A -85,B 0,C 180,E1 -20626.608,E2 -20626.608} C_VEL
LIN {X 0,Y 217.203,Z 376.374,A -85,B 0,C 180,E1 -20629.369,E2 -20629.369} C_VEL
LIN {X 0,Y 219.298,Z 369.041,A -85,B 0,C 180,E1 -20631.802,E2 -20631.802} C_VEL
LIN {X 0,Y 222.032,Z 359.583,A -85,B 0,C 180,E1 -20634.298,E2 -20634.298} C_VEL
LIN {X 0,Y 224.843,Z 349.082,A -85,B 0,C 180,E1 -20636.45,E2 -20636.45} C_VEL
LIN {X 0,Y 227.697,Z 337.262,A -85,B 0,C 180,E1 -20638.331,E2 -20638.331} C_VEL
LIN {X 0,Y 230.024,Z 325.346,A -85,B 0,C 180,E1 -20639.768,E2 -20639.768} C_VEL
LIN {X 0,Y 232.054,Z 312.944,A -85,B 0,C 180,E1 -20640.862,E2 -20640.862} C_VEL
LIN {X 0,Y 233.6,Z 300.29,A -85,B 0,C 180,E1 -20641.633,E2 -20641.633} C_VEL
LIN {X 0,Y 234.474,Z 286.53,A -85,B 0,C 180,E1 -20642.144,E2 -20642.144} C_VEL
LIN {X 0,Y 236.207,Z 240.185,A -85,B 0,C 180,E1 -20643.519,E2 -20643.519} C_VEL
LIN {X 0,Y 234.095,Z 225.775,A -85,B 0,C 180,E1 -20644.381,E2 -20644.381} C_VEL
LIN {X 0,Y 227.041,Z 208.825,A -85,B 0,C 180,E1 -20646.247,E2 -20646.247} C_VEL
LIN {X 0,Y 220.413,Z 195.368,A -85,B 0,C 180,E1 -20648.054,E2 -20648.054} C_VEL
LIN {X 0,Y 215.628,Z 186.387,A -85,B 0,C 180,E1 -20649.462,E2 -20649.462} C_VEL
LIN {X 0,Y 213.712,Z 179.366,A -85,B 0,C 180,E1 -20653.499,E2 -20653.499} C_VEL
LIN {X 0,Y 213.703,Z 179.366,A -85,B 0,C 180,E1 -20656.345,E2 -20656.345} C_VEL
LIN {X 0,Y 213.716,Z 179.363,A -85,B 0,C 180,E1 -20659.143,E2 -20659.143} C_VEL
LIN {X 0,Y 213.744,Z 179.36,A -85,B 0,C 180,E1 -20663.712,E2 -20663.712} C_VEL
LIN {X 0,Y 213.759,Z 179.359,A -85,B 0,C 180,E1 -20668.261,E2 -20668.261} C_VEL
LIN {X 0,Y 213.789,Z 179.347,A -85,B 0,C 180,E1 -20672.598,E2 -20672.598} C_VEL
LIN {X 0,Y 213.812,Z 179.344,A -85,B 0,C 180,E1 -20676.978,E2 -20676.978} C_VEL
LIN {X 0,Y 213.944,Z 179.327,A -85,B 0,C 180,E1 -20682.804,E2 -20682.804} C_VEL
LIN {X 0,Y 213.954,Z 179.328,A -85,B 0,C 180,E1 -20686.707,E2 -20686.707} C_VEL
LIN {X 0,Y 214.143,Z 179.31,A -85,B 0,C 180,E1 -20690.555,E2 -20690.555} C_VEL
LIN {X 0,Y 214.101,Z 179.308,A -85,B 0,C 180,E1 -20694.349,E2 -20694.349} C_VEL
LIN {X 0,Y 214.446,Z 179.268,A -85,B 0,C 180,E1 -20698.122,E2 -20698.122} C_VEL
LIN {X 0,Y 214.547,Z 179.25,A -85,B 0,C 180,E1 -20700,E2 -20700} C_VEL
LIN {X 0,Y 214.445,Z 179.272,A -85,B 0,C 180,E1 -20701.878,E2 -20701.878} C_VEL
LIN {X 0,Y 214.199,Z 179.303,A -85,B 0,C 180,E1 -20707.542,E2 -20707.542} C_VEL
LIN {X 0,Y 214,Z 179.317,A -85,B 0,C 180,E1 -20711.364,E2 -20711.364} C_VEL
LIN {X 0,Y 213.935,Z 179.335,A -85,B 0,C 180,E1 -20715.237,E2 -20715.237} C_VEL
LIN {X 0,Y 213.869,Z 179.345,A -85,B 0,C 180,E1 -20719.185,E2 -20719.185} C_VEL
LIN {X 0,Y 213.848,Z 179.34,A -85,B 0,C 180,E1 -20723.227,E2 -20723.227} C_VEL
LIN {X 0,Y 213.83,Z 179.34,A -85,B 0,C 180,E1 -20727.45,E2 -20727.45} C_VEL
LIN {X 0,Y 213.78,Z 179.349,A -85,B 0,C 180,E1 -20731.736,E2 -20731.736} C_VEL
LIN {X 0,Y 213.753,Z 179.354,A -85,B 0,C 180,E1 -20736.287,E2 -20736.287} C_VEL
LIN {X 0,Y 213.718,Z 179.364,A -85,B 0,C 180,E1 -20741.124,E2 -20741.124} C_VEL
LIN {X 0,Y 213.708,Z 179.364,A -85,B 0,C 180,E1 -20743.678,E2 -20743.678} C_VEL
LIN {X 0,Y 213.707,Z 179.364,A -85,B 0,C 180,E1 -20746.344,E2 -20746.344} C_VEL
LIN {X 0,Y 213.761,Z 179.355,A -85,B 0,C 180,E1 -20750.207,E2 -20750.207} C_VEL
LIN {X 0,Y 214.787,Z 182.251,A -85,B 0,C 180,E1 -20750.58,E2 -20750.58} C_VEL
LIN {X 0,Y 216.527,Z 184.538,A -85,B 0,C 180,E1 -20751.056,E2 -20751.056} C_VEL
LIN {X 0,Y 221.483,Z 192.745,A -85,B 0,C 180,E1 -20752.422,E2 -20752.422} C_VEL
LIN {X 0,Y 228.304,Z 206.081,A -85,B 0,C 180,E1 -20754.246,E2 -20754.246} C_VEL
LIN {X 0,Y 234.46,Z 220.046,A -85,B 0,C 180,E1 -20755.838,E2 -20755.838} C_VEL
LIN {X 0,Y 236.842,Z 226.219,A -85,B 0,C 180,E1 -20756.451,E2 -20756.451} C_VEL
LIN {X 0,Y 234.534,Z 283.102,A -85,B 0,C 180,E1 -20758.131,E2 -20758.131} C_VEL
LIN {X 0,Y 233.511,Z 296.121,A -85,B 0,C 180,E1 -20758.739,E2 -20758.739} C_VEL
LIN {X 0,Y 231.958,Z 308.395,A -85,B 0,C 180,E1 -20759.628,E2 -20759.628} C_VEL
LIN {X 0,Y 229.822,Z 321.356,A -85,B 0,C 180,E1 -20760.957,E2 -20760.957} C_VEL
LIN {X 0,Y 227.585,Z 332.099,A -85,B 0,C 180,E1 -20762.406,E2 -20762.406} C_VEL
LIN {X 0,Y 224.951,Z 343.047,A -85,B 0,C 180,E1 -20764.311,E2 -20764.311} C_VEL
LIN {X 0,Y 222.353,Z 353.125,A -85,B 0,C 180,E1 -20766.564,E2 -20766.564} C_VEL
LIN {X 0,Y 219.985,Z 361.58,A -85,B 0,C 180,E1 -20768.936,E2 -20768.936} C_VEL
LIN {X 0,Y 217.447,Z 369.27,A -85,B 0,C 180,E1 -20771.632,E2 -20771.632} C_VEL
LIN {X 0,Y 215.225,Z 376.326,A -85,B 0,C 180,E1 -20774.857,E2 -20774.857} C_VEL
LIN {X 0,Y 213.713,Z 381.024,A -85,B 0,C 180,E1 -20777.658,E2 -20777.658} C_VEL
LIN {X 0,Y 212.679,Z 384.617,A -85,B 0,C 180,E1 -20780.49,E2 -20780.49} C_VEL
LIN {X 0,Y 212.234,Z 386.471,A -85,B 0,C 180,E1 -20782.388,E2 -20782.388} C_VEL
LIN {X 0,Y 211.831,Z 387.964,A -85,B 0,C 180,E1 -20784.458,E2 -20784.458} C_VEL
LIN {X 0,Y 211.546,Z 389.465,A -85,B 0,C 180,E1 -20788.096,E2 -20788.096} C_VEL
LIN {X 0,Y 211.522,Z 389.694,A -85,B 0,C 180,E1 -20790,E2 -20790} C_VEL
LIN {X 0,Y 211.545,Z 389.5,A -85,B 0,C 180,E1 -20791.904,E2 -20791.904} C_VEL
LIN {X 0,Y 211.853,Z 387.945,A -85,B 0,C 180,E1 -20795.712,E2 -20795.712} C_VEL
LIN {X 0,Y 212.162,Z 386.587,A -85,B 0,C 180,E1 -20797.614,E2 -20797.614} C_VEL
LIN {X 0,Y 212.951,Z 383.715,A -85,B 0,C 180,E1 -20800.458,E2 -20800.458} C_VEL
LIN {X 0,Y 214.134,Z 379.82,A -85,B 0,C 180,E1 -20803.282,E2 -20803.282} C_VEL
LIN {X 0,Y 215.748,Z 374.794,A -85,B 0,C 180,E1 -20806.074,E2 -20806.074} C_VEL
LIN {X 0,Y 217.805,Z 368.462,A -85,B 0,C 180,E1 -20808.825,E2 -20808.825} C_VEL
LIN {X 0,Y 220.362,Z 360.537,A -85,B 0,C 180,E1 -20811.516,E2 -20811.516} C_VEL
LIN {X 0,Y 222.696,Z 351.954,A -85,B 0,C 180,E1 -20813.868,E2 -20813.868} C_VEL
LIN {X 0,Y 225.471,Z 341.507,A -85,B 0,C 180,E1 -20816.122,E2 -20816.122} C_VEL
LIN {X 0,Y 227.856,Z 331.507,A -85,B 0,C 180,E1 -20817.808,E2 -20817.808} C_VEL
LIN {X 0,Y 230.071,Z 320.624,A -85,B 0,C 180,E1 -20819.259,E2 -20819.259} C_VEL
LIN {X 0,Y 232.073,Z 308.593,A -85,B 0,C 180,E1 -20820.481,E2 -20820.481} C_VEL
LIN {X 0,Y 233.553,Z 296.04,A -85,B 0,C 180,E1 -20821.409,E2 -20821.409} C_VEL
LIN {X 0,Y 234.636,Z 282.968,A -85,B 0,C 180,E1 -20822.006,E2 -20822.006} C_VEL
LIN {X 0,Y 237.023,Z 226.509,A -85,B 0,C 180,E1 -20823.657,E2 -20823.657} C_VEL
LIN {X 0,Y 232.732,Z 215.816,A -85,B 0,C 180,E1 -20824.76,E2 -20824.76} C_VEL
LIN {X 0,Y 226.003,Z 201.354,A -85,B 0,C 180,E1 -20826.518,E2 -20826.518} C_VEL
LIN {X 0,Y 219.852,Z 189.82,A -85,B 0,C 180,E1 -20828.19,E2 -20828.19} C_VEL
LIN {X 0,Y 216.443,Z 184.259,A -85,B 0,C 180,E1 -20829.14,E2 -20829.14} C_VEL
LIN {X 0,Y 214.345,Z 181.373,A -85,B 0,C 180,E1 -20829.723,E2 -20829.723} C_VEL
LIN {X 0,Y 213.762,Z 179.355,A -85,B 0,C 180,E1 -20829.956,E2 -20829.956} C_VEL
LIN {X 0,Y 213.707,Z 179.365,A -85,B 0,C 180,E1 -20833.678,E2 -20833.678} C_VEL
LIN {X 0,Y 213.708,Z 179.366,A -85,B 0,C 180,E1 -20836.343,E2 -20836.343} C_VEL
LIN {X 0,Y 213.736,Z 179.354,A -85,B 0,C 180,E1 -20841.336,E2 -20841.336} C_VEL
LIN {X 0,Y 213.768,Z 179.346,A -85,B 0,C 180,E1 -20846.02,E2 -20846.02} C_VEL
LIN {X 0,Y 213.781,Z 179.351,A -85,B 0,C 180,E1 -20850.454,E2 -20850.454} C_VEL
LIN {X 0,Y 213.802,Z 179.352,A -85,B 0,C 180,E1 -20854.702,E2 -20854.702} C_VEL
LIN {X 0,Y 213.813,Z 179.341,A -85,B 0,C 180,E1 -20858.803,E2 -20858.803} C_VEL
LIN {X 0,Y 213.944,Z 179.328,A -85,B 0,C 180,E1 -20862.803,E2 -20862.803} C_VEL
LIN {X 0,Y 213.981,Z 179.327,A -85,B 0,C 180,E1 -20866.708,E2 -20866.708} C_VEL
LIN {X 0,Y 214.167,Z 179.294,A -85,B 0,C 180,E1 -20870.556,E2 -20870.556} C_VEL
LIN {X 0,Y 214.227,Z 179.287,A -85,B 0,C 180,E1 -20872.459,E2 -20872.459} C_VEL
LIN {X 0,Y 214.446,Z 179.258,A -85,B 0,C 180,E1 -20878.122,E2 -20878.122} C_VEL
LIN {X 0,Y 214.546,Z 179.249,A -85,B 0,C 180,E1 -20880,E2 -20880} C_VEL
LIN {X 0,Y 214.446,Z 179.271,A -85,B 0,C 180,E1 -20881.878,E2 -20881.878} C_VEL
LIN {X 0,Y 214.227,Z 179.291,A -85,B 0,C 180,E1 -20887.54,E2 -20887.54} C_VEL
LIN {X 0,Y 214.023,Z 179.32,A -85,B 0,C 180,E1 -20891.363,E2 -20891.363} C_VEL
LIN {X 0,Y 213.934,Z 179.333,A -85,B 0,C 180,E1 -20895.237,E2 -20895.237} C_VEL
LIN {X 0,Y 213.835,Z 179.334,A -85,B 0,C 180,E1 -20899.188,E2 -20899.188} C_VEL
LIN {X 0,Y 213.811,Z 179.35,A -85,B 0,C 180,E1 -20903.231,E2 -20903.231} C_VEL
LIN {X 0,Y 213.829,Z 179.349,A -85,B 0,C 180,E1 -20907.45,E2 -20907.45} C_VEL
LIN {X 0,Y 213.767,Z 179.355,A -85,B 0,C 180,E1 -20911.738,E2 -20911.738} C_VEL
LIN {X 0,Y 213.744,Z 179.361,A -85,B 0,C 180,E1 -20916.288,E2 -20916.288} C_VEL
LIN {X 0,Y 213.711,Z 179.361,A -85,B 0,C 180,E1 -20921.126,E2 -20921.126} C_VEL
LIN {X 0,Y 213.667,Z 179.363,A -85,B 0,C 180,E1 -20924.187,E2 -20924.187} C_VEL
LIN {X 0,Y 212.926,Z 179.837,A -85,B 0,C 180,E1 -20925.307,E2 -20925.307} C_VEL
LIN {X 0,Y 210.831,Z 181.615,A -85,B 0,C 180,E1 -20926.687,E2 -20926.687} C_VEL
LIN {X 0,Y 209.054,Z 184.35,A -85,B 0,C 180,E1 -20927.932,E2 -20927.932} C_VEL
LIN {X 0,Y 208.786,Z 186.975,A -85,B 0,C 180,E1 -20928.773,E2 -20928.773} C_VEL
LIN {X 0,Y 209.537,Z 188.878,A -85,B 0,C 180,E1 -20929.227,E2 -20929.227} C_VEL
LIN {X 0,Y 211.699,Z 192.506,A -85,B 0,C 180,E1 -20929.884,E2 -20929.884} C_VEL
LIN {X 0,Y 216.591,Z 201.479,A -85,B 0,C 180,E1 -20931.334,E2 -20931.334} C_VEL
LIN {X 0,Y 222.944,Z 214.778,A -85,B 0,C 180,E1 -20933.148,E2 -20933.148} C_VEL
LIN {X 0,Y 228.746,Z 229.117,A -85,B 0,C 180,E1 -20934.765,E2 -20934.765} C_VEL
LIN {X 0,Y 230.455,Z 242.673,A -85,B 0,C 180,E1 -20935.566,E2 -20935.566} C_VEL
LIN {X 0,Y 228.082,Z 295.248,A -85,B 0,C 180,E1 -20937.164,E2 -20937.164} C_VEL
LIN {X 0,Y 226.678,Z 308.822,A -85,B 0,C 180,E1 -20937.895,E2 -20937.895} C_VEL
LIN {X 0,Y 224.861,Z 320.548,A -85,B 0,C 180,E1 -20938.825,E2 -20938.825} C_VEL
LIN {X 0,Y 222.589,Z 332.739,A -85,B 0,C 180,E1 -20940.179,E2 -20940.179} C_VEL
LIN {X 0,Y 219.857,Z 344.293,A -85,B 0,C 180,E1 -20941.868,E2 -20941.868} C_VEL
LIN {X 0,Y 217.028,Z 354.7,A -85,B 0,C 180,E1 -20943.819,E2 -20943.819} C_VEL
LIN {X 0,Y 214.518,Z 363.21,A -85,B 0,C 180,E1 -20945.825,E2 -20945.825} C_VEL
LIN {X 0,Y 212.139,Z 371.497,A -85,B 0,C 180,E1 -20948.274,E2 -20948.274} C_VEL
LIN {X 0,Y 209.706,Z 378.737,A -85,B 0,C 180,E1 -20950.928,E2 -20950.928} C_VEL
LIN {X 0,Y 208.037,Z 383.998,A -85,B 0,C 180,E1 -20953.313,E2 -20953.313} C_VEL
LIN {X 0,Y 206.357,Z 389.094,A -85,B 0,C 180,E1 -20956.208,E2 -20956.208} C_VEL
LIN {X 0,Y 205.309,Z 393.056,A -85,B 0,C 180,E1 -20959.148,E2 -20959.148} C_VEL
LIN {X 0,Y 204.626,Z 395.985,A -85,B 0,C 180,E1 -20962.104,E2 -20962.104} C_VEL
LIN {X 0,Y 204.297,Z 398.375,A -85,B 0,C 180,E1 -20966.055,E2 -20966.055} C_VEL
LIN {X 0,Y 204.325,Z 398.983,A -85,B 0,C 180,E1 -20968.029,E2 -20968.029} C_VEL
LIN {X 0,Y 204.392,Z 399.196,A -85,B 0,C 180,E1 -20970,E2 -20970} C_VEL
LIN {X 0,Y 204.325,Z 398.97,A -85,B 0,C 180,E1 -20971.971,E2 -20971.971} C_VEL
LIN {X 0,Y 204.297,Z 398.354,A -85,B 0,C 180,E1 -20973.945,E2 -20973.945} C_VEL
LIN {X 0,Y 204.398,Z 397.351,A -85,B 0,C 180,E1 -20975.921,E2 -20975.921} C_VEL
LIN {X 0,Y 204.626,Z 395.944,A -85,B 0,C 180,E1 -20977.896,E2 -20977.896} C_VEL
LIN {X 0,Y 205.309,Z 392.997,A -85,B 0,C 180,E1 -20980.852,E2 -20980.852} C_VEL
LIN {X 0,Y 206.356,Z 389.012,A -85,B 0,C 180,E1 -20983.792,E2 -20983.792} C_VEL
LIN {X 0,Y 208.337,Z 382.892,A -85,B 0,C 180,E1 -20987.168,E2 -20987.168} C_VEL
LIN {X 0,Y 210.509,Z 376.21,A -85,B 0,C 180,E1 -20990.011,E2 -20990.011} C_VEL
LIN {X 0,Y 213.046,Z 367.82,A -85,B 0,C 180,E1 -20992.84,E2 -20992.84} C_VEL
LIN {X 0,Y 215.576,Z 359.418,A -85,B 0,C 180,E1 -20995.076,E2 -20995.076} C_VEL
LIN {X 0,Y 218.501,Z 348.916,A -85,B 0,C 180,E1 -20997.28,E2 -20997.28} C_VEL
LIN {X 0,Y 221.468,Z 337.095,A -85,B 0,C 180,E1 -20999.203,E2 -20999.203} C_VEL
LIN {X 0,Y 223.897,Z 325.178,A -85,B 0,C 180,E1 -21000.669,E2 -21000.669} C_VEL
LIN {X 0,Y 226.004,Z 312.774,A -85,B 0,C 180,E1 -21001.783,E2 -21001.783} C_VEL
LIN {X 0,Y 227.631,Z 299.775,A -85,B 0,C 180,E1 -21002.586,E2 -21002.586} C_VEL
LIN {X 0,Y 228.591,Z 284.874,A -85,B 0,C 180,E1 -21003.129,E2 -21003.129} C_VEL
LIN {X 0,Y 230.29,Z 241.304,A -85,B 0,C 180,E1 -21004.451,E2 -21004.451} C_VEL
LIN {X 0,Y 228.462,Z 228.418,A -85,B 0,C 180,E1 -21005.247,E2 -21005.247} C_VEL
LIN {X 0,Y 221.385,Z 211.352,A -85,B 0,C 180,E1 -21007.22,E2 -21007.22} C_VEL
LIN {X 0,Y 215.57,Z 199.53,A -85,B 0,C 180,E1 -21008.888,E2 -21008.888} C_VEL
LIN {X 0,Y 210.203,Z 189.916,A -85,B 0,C 180,E1 -21010.491,E2 -21010.491} C_VEL
LIN {X 0,Y 208.257,Z 186.103,A -85,B 0,C 180,E1 -21011.185,E2 -21011.185} C_VEL
LIN {X 0,Y 206.604,Z 180.251,A -85,B 0,C 180,E1 -21014.745,E2 -21014.745} C_VEL
LIN {X 0,Y 206.66,Z 180.243,A -85,B 0,C 180,E1 -21019.749,E2 -21019.749} C_VEL
LIN {X 0,Y 206.699,Z 180.239,A -85,B 0,C 180,E1 -21024.689,E2 -21024.689} C_VEL
LIN {X 0,Y 206.696,Z 180.238,A -85,B 0,C 180,E1 -21029.334,E2 -21029.334} C_VEL
LIN {X 0,Y 206.706,Z 180.232,A -85,B 0,C 180,E1 -21033.769,E2 -21033.769} C_VEL
LIN {X 0,Y 206.738,Z 180.226,A -85,B 0,C 180,E1 -21038.041,E2 -21038.041} C_VEL
LIN {X 0,Y 206.873,Z 180.206,A -85,B 0,C 180,E1 -21042.197,E2 -21042.197} C_VEL
LIN {X 0,Y 206.896,Z 180.209,A -85,B 0,C 180,E1 -21046.244,E2 -21046.244} C_VEL
LIN {X 0,Y 207.1,Z 180.188,A -85,B 0,C 180,E1 -21050.231,E2 -21050.231} C_VEL
LIN {X 0,Y 207.062,Z 180.183,A -85,B 0,C 180,E1 -21054.156,E2 -21054.156} C_VEL
LIN {X 0,Y 207.383,Z 180.147,A -85,B 0,C 180,E1 -21058.058,E2 -21058.058} C_VEL
LIN {X 0,Y 207.512,Z 180.126,A -85,B 0,C 180,E1 -21060,E2 -21060} C_VEL
LIN {X 0,Y 207.382,Z 180.152,A -85,B 0,C 180,E1 -21061.942,E2 -21061.942} C_VEL
LIN {X 0,Y 207.141,Z 180.182,A -85,B 0,C 180,E1 -21067.8,E2 -21067.8} C_VEL
LIN {X 0,Y 206.925,Z 180.198,A -85,B 0,C 180,E1 -21071.758,E2 -21071.758} C_VEL
LIN {X 0,Y 206.868,Z 180.214,A -85,B 0,C 180,E1 -21075.771,E2 -21075.771} C_VEL
LIN {X 0,Y 206.8,Z 180.225,A -85,B 0,C 180,E1 -21079.868,E2 -21079.868} C_VEL
LIN {X 0,Y 206.765,Z 180.225,A -85,B 0,C 180,E1 -21084.072,E2 -21084.072} C_VEL
LIN {X 0,Y 206.745,Z 180.225,A -85,B 0,C 180,E1 -21088.419,E2 -21088.419} C_VEL
LIN {X 0,Y 206.71,Z 180.233,A -85,B 0,C 180,E1 -21092.956,E2 -21092.956} C_VEL
LIN {X 0,Y 206.723,Z 180.231,A -85,B 0,C 180,E1 -21095.32,E2 -21095.32} C_VEL
LIN {X 0,Y 206.668,Z 180.24,A -85,B 0,C 180,E1 -21100.25,E2 -21100.25} C_VEL
LIN {X 0,Y 206.635,Z 180.241,A -85,B 0,C 180,E1 -21105.582,E2 -21105.582} C_VEL
LIN {X 0,Y 206.662,Z 180.24,A -85,B 0,C 180,E1 -21108.577,E2 -21108.577} C_VEL
LIN {X 0,Y 207.692,Z 183.122,A -85,B 0,C 180,E1 -21108.98,E2 -21108.98} C_VEL
LIN {X 0,Y 209.63,Z 185.527,A -85,B 0,C 180,E1 -21109.549,E2 -21109.549} C_VEL
LIN {X 0,Y 216.483,Z 196.512,A -85,B 0,C 180,E1 -21111.546,E2 -21111.546} C_VEL
LIN {X 0,Y 223.458,Z 210.453,A -85,B 0,C 180,E1 -21113.511,E2 -21113.511} C_VEL
LIN {X 0,Y 229.572,Z 224.524,A -85,B 0,C 180,E1 -21115.168,E2 -21115.168} C_VEL
LIN {X 0,Y 230.916,Z 228.094,A -85,B 0,C 180,E1 -21115.533,E2 -21115.533} C_VEL
LIN {X 0,Y 228.478,Z 284.392,A -85,B 0,C 180,E1 -21117.23,E2 -21117.23} C_VEL
LIN {X 0,Y 227.369,Z 297.208,A -85,B 0,C 180,E1 -21117.867,E2 -21117.867} C_VEL
LIN {X 0,Y 225.685,Z 309.692,A -85,B 0,C 180,E1 -21118.821,E2 -21118.821} C_VEL
LIN {X 0,Y 223.653,Z 321.524,A -85,B 0,C 180,E1 -21120.076,E2 -21120.076} C_VEL
LIN {X 0,Y 221.335,Z 332.265,A -85,B 0,C 180,E1 -21121.557,E2 -21121.557} C_VEL
LIN {X 0,Y 218.565,Z 343.213,A -85,B 0,C 180,E1 -21123.503,E2 -21123.503} C_VEL
LIN {X 0,Y 215.853,Z 353.29,A -85,B 0,C 180,E1 -21125.814,E2 -21125.814} C_VEL
LIN {X 0,Y 213.385,Z 361.745,A -85,B 0,C 180,E1 -21128.252,E2 -21128.252} C_VEL
LIN {X 0,Y 210.729,Z 369.434,A -85,B 0,C 180,E1 -21131.024,E2 -21131.024} C_VEL
LIN {X 0,Y 208.982,Z 374.681,A -85,B 0,C 180,E1 -21133.39,E2 -21133.39} C_VEL
LIN {X 0,Y 207.268,Z 379.77,A -85,B 0,C 180,E1 -21136.27,E2 -21136.27} C_VEL
LIN {X 0,Y 206.001,Z 383.719,A -85,B 0,C 180,E1 -21139.185,E2 -21139.185} C_VEL
LIN {X 0,Y 205.192,Z 386.634,A -85,B 0,C 180,E1 -21142.125,E2 -21142.125} C_VEL
LIN {X 0,Y 204.697,Z 388.358,A -85,B 0,C 180,E1 -21144.674,E2 -21144.674} C_VEL
LIN {X 0,Y 204.452,Z 389.627,A -85,B 0,C 180,E1 -21148.03,E2 -21148.03} C_VEL
LIN {X 0,Y 204.424,Z 389.856,A -85,B 0,C 180,E1 -21150,E2 -21150} C_VEL
LIN {X 0,Y 204.451,Z 389.662,A -85,B 0,C 180,E1 -21151.97,E2 -21151.97} C_VEL
LIN {X 0,Y 204.693,Z 388.445,A -85,B 0,C 180,E1 -21155.313,E2 -21155.313} C_VEL
LIN {X 0,Y 205.12,Z 386.749,A -85,B 0,C 180,E1 -21157.877,E2 -21157.877} C_VEL
LIN {X 0,Y 205.96,Z 383.877,A -85,B 0,C 180,E1 -21160.817,E2 -21160.817} C_VEL
LIN {X 0,Y 207.236,Z 379.981,A -85,B 0,C 180,E1 -21163.732,E2 -21163.732} C_VEL
LIN {X 0,Y 208.922,Z 374.955,A -85,B 0,C 180,E1 -21166.615,E2 -21166.615} C_VEL
LIN {X 0,Y 211.089,Z 368.622,A -85,B 0,C 180,E1 -21169.447,E2 -21169.447} C_VEL
LIN {X 0,Y 213.764,Z 360.697,A -85,B 0,C 180,E1 -21172.215,E2 -21172.215} C_VEL
LIN {X 0,Y 216.134,Z 352.387,A -85,B 0,C 180,E1 -21174.562,E2 -21174.562} C_VEL
LIN {X 0,Y 218.829,Z 342.766,A -85,B 0,C 180,E1 -21176.72,E2 -21176.72} C_VEL
LIN {X 0,Y 221.305,Z 333.059,A -85,B 0,C 180,E1 -21178.447,E2 -21178.447} C_VEL
LIN {X 0,Y 223.573,Z 322.542,A -85,B 0,C 180,E1 -21179.936,E2 -21179.936} C_VEL
LIN {X 0,Y 225.815,Z 309.876,A -85,B 0,C 180,E1 -21181.289,E2 -21181.289} C_VEL
LIN {X 0,Y 227.421,Z 297.223,A -85,B 0,C 180,E1 -21182.275,E2 -21182.275} C_VEL
LIN {X 0,Y 228.616,Z 284.294,A -85,B 0,C 180,E1 -21182.903,E2 -21182.903} C_VEL
LIN {X 0,Y 231.067,Z 228.36,A -85,B 0,C 180,E1 -21184.583,E2 -21184.583} C_VEL
LIN {X 0,Y 226.02,Z 215.95,A -85,B 0,C 180,E1 -21185.951,E2 -21185.951} C_VEL
LIN {X 0,Y 218.392,Z 200.091,A -85,B 0,C 180,E1 -21188.071,E2 -21188.071} C_VEL
LIN {X 0,Y 213.853,Z 192.18,A -85,B 0,C 180,E1 -21189.371,E2 -21189.371} C_VEL
LIN {X 0,Y 209.559,Z 185.331,A -85,B 0,C 180,E1 -21190.649,E2 -21190.649} C_VEL
LIN {X 0,Y 207.288,Z 182.36,A -85,B 0,C 180,E1 -21191.327,E2 -21191.327} C_VEL
LIN {X 0,Y 206.651,Z 180.241,A -85,B 0,C 180,E1 -21191.621,E2 -21191.621} C_VEL
LIN {X 0,Y 206.635,Z 180.242,A -85,B 0,C 180,E1 -21195.581,E2 -21195.581} C_VEL
LIN {X 0,Y 206.667,Z 180.24,A -85,B 0,C 180,E1 -21199.75,E2 -21199.75} C_VEL
LIN {X 0,Y 206.732,Z 180.231,A -85,B 0,C 180,E1 -21204.695,E2 -21204.695} C_VEL
LIN {X 0,Y 206.724,Z 180.234,A -85,B 0,C 180,E1 -21209.339,E2 -21209.339} C_VEL
LIN {X 0,Y 206.734,Z 180.23,A -85,B 0,C 180,E1 -21213.772,E2 -21213.772} C_VEL
LIN {X 0,Y 206.757,Z 180.216,A -85,B 0,C 180,E1 -21218.043,E2 -21218.043} C_VEL
LIN {X 0,Y 206.874,Z 180.213,A -85,B 0,C 180,E1 -21222.196,E2 -21222.196} C_VEL
LIN {X 0,Y 206.914,Z 180.206,A -85,B 0,C 180,E1 -21226.245,E2 -21226.245} C_VEL
LIN {X 0,Y 207.105,Z 180.176,A -85,B 0,C 180,E1 -21230.231,E2 -21230.231} C_VEL
LIN {X 0,Y 207.167,Z 180.164,A -85,B 0,C 180,E1 -21232.201,E2 -21232.201} C_VEL
LIN {X 0,Y 207.382,Z 180.137,A -85,B 0,C 180,E1 -21238.058,E2 -21238.058} C_VEL
LIN {X 0,Y 207.512,Z 180.124,A -85,B 0,C 180,E1 -21240,E2 -21240} C_VEL
LIN {X 0,Y 207.382,Z 180.151,A -85,B 0,C 180,E1 -21241.942,E2 -21241.942} C_VEL
LIN {X 0,Y 207.167,Z 180.172,A -85,B 0,C 180,E1 -21247.799,E2 -21247.799} C_VEL
LIN {X 0,Y 206.943,Z 180.197,A -85,B 0,C 180,E1 -21251.757,E2 -21251.757} C_VEL
LIN {X 0,Y 206.867,Z 180.214,A -85,B 0,C 180,E1 -21255.771,E2 -21255.771} C_VEL
LIN {X 0,Y 206.763,Z 180.215,A -85,B 0,C 180,E1 -21259.871,E2 -21259.871} C_VEL
LIN {X 0,Y 206.747,Z 180.223,A -85,B 0,C 180,E1 -21264.074,E2 -21264.074} C_VEL
LIN {X 0,Y 206.737,Z 180.232,A -85,B 0,C 180,E1 -21268.42,E2 -21268.42} C_VEL
LIN {X 0,Y 206.699,Z 180.238,A -85,B 0,C 180,E1 -21272.958,E2 -21272.958} C_VEL
LIN {X 0,Y 206.679,Z 180.235,A -85,B 0,C 180,E1 -21277.74,E2 -21277.74} C_VEL
LIN {X 0,Y 206.64,Z 180.24,A -85,B 0,C 180,E1 -21281.562,E2 -21281.562} C_VEL
LIN {X 0,Y 206.607,Z 180.257,A -85,B 0,C 180,E1 -21285.254,E2 -21285.254} C_VEL
LIN {X 0,Y 208.383,Z 186.49,A -85,B 0,C 180,E1 -21288.847,E2 -21288.847} C_VEL
LIN {X 0,Y 209.537,Z 188.878,A -85,B 0,C 180,E1 -21289.227,E2 -21289.227} C_VEL
LIN {X 0,Y 210.906,Z 192.157,A -85,B 0,C 180,E1 -21289.688,E2 -21289.688} C_VEL
LIN {X 0,Y 211.731,Z 198.576,A -85,B 0,C 180,E1 -21290.154,E2 -21290.154} C_VEL
LIN {X 0,Y 212.338,Z 205.202,A -85,B 0,C 180,E1 -21290.574,E2 -21290.574} C_VEL
LIN {X 0,Y 213.423,Z 208.813,A -85,B 0,C 180,E1 -21290.965,E2 -21290.965} C_VEL
LIN {X 0,Y 219.973,Z 223.509,A -85,B 0,C 180,E1 -21292.919,E2 -21292.919} C_VEL
LIN {X 0,Y 223.217,Z 232.24,A -85,B 0,C 180,E1 -21293.884,E2 -21293.884} C_VEL
LIN {X 0,Y 224.593,Z 243.572,A -85,B 0,C 180,E1 -21294.574,E2 -21294.574} C_VEL
LIN {X 0,Y 222.163,Z 294.928,A -85,B 0,C 180,E1 -21296.164,E2 -21296.164} C_VEL
LIN {X 0,Y 220.691,Z 308.801,A -85,B 0,C 180,E1 -21296.926,E2 -21296.926} C_VEL
LIN {X 0,Y 218.823,Z 320.393,A -85,B 0,C 180,E1 -21297.863,E2 -21297.863} C_VEL
LIN {X 0,Y 216.458,Z 332.581,A -85,B 0,C 180,E1 -21299.245,E2 -21299.245} C_VEL
LIN {X 0,Y 213.603,Z 344.135,A -85,B 0,C 180,E1 -21300.968,E2 -21300.968} C_VEL
LIN {X 0,Y 210.667,Z 354.541,A -85,B 0,C 180,E1 -21302.965,E2 -21302.965} C_VEL
LIN {X 0,Y 208.053,Z 363.05,A -85,B 0,C 180,E1 -21305.024,E2 -21305.024} C_VEL
LIN {X 0,Y 205.633,Z 370.768,A -85,B 0,C 180,E1 -21307.338,E2 -21307.338} C_VEL
LIN {X 0,Y 202.979,Z 378.576,A -85,B 0,C 180,E1 -21310.27,E2 -21310.27} C_VEL
LIN {X 0,Y 201.2,Z 383.836,A -85,B 0,C 180,E1 -21312.728,E2 -21312.728} C_VEL
LIN {X 0,Y 199.428,Z 388.931,A -85,B 0,C 180,E1 -21315.719,E2 -21315.719} C_VEL
LIN {X 0,Y 198.297,Z 392.894,A -85,B 0,C 180,E1 -21318.76,E2 -21318.76} C_VEL
LIN {X 0,Y 197.58,Z 395.823,A -85,B 0,C 180,E1 -21321.82,E2 -21321.82} C_VEL
LIN {X 0,Y 197.206,Z 398.212,A -85,B 0,C 180,E1 -21325.913,E2 -21325.913} C_VEL
LIN {X 0,Y 197.232,Z 398.821,A -85,B 0,C 180,E1 -21327.958,E2 -21327.958} C_VEL
LIN {X 0,Y 197.296,Z 399.033,A -85,B 0,C 180,E1 -21330,E2 -21330} C_VEL
LIN {X 0,Y 197.201,Z 398.335,A -85,B 0,C 180,E1 -21333.724,E2 -21333.724} C_VEL
LIN {X 0,Y 197.338,Z 397.188,A -85,B 0,C 180,E1 -21336.133,E2 -21336.133} C_VEL
LIN {X 0,Y 197.58,Z 395.781,A -85,B 0,C 180,E1 -21338.18,E2 -21338.18} C_VEL
LIN {X 0,Y 198.297,Z 392.833,A -85,B 0,C 180,E1 -21341.241,E2 -21341.241} C_VEL
LIN {X 0,Y 199.427,Z 388.848,A -85,B 0,C 180,E1 -21344.282,E2 -21344.282} C_VEL
LIN {X 0,Y 201.552,Z 382.728,A -85,B 0,C 180,E1 -21347.765,E2 -21347.765} C_VEL
LIN {X 0,Y 203.847,Z 376.045,A -85,B 0,C 180,E1 -21350.695,E2 -21350.695} C_VEL
LIN {X 0,Y 206.413,Z 367.902,A -85,B 0,C 180,E1 -21353.529,E2 -21353.529} C_VEL
LIN {X 0,Y 209.14,Z 359.252,A -85,B 0,C 180,E1 -21355.903,E2 -21355.903} C_VEL
LIN {X 0,Y 212.225,Z 348.751,A -85,B 0,C 180,E1 -21358.158,E2 -21358.158} C_VEL
LIN {X 0,Y 215.282,Z 336.928,A -85,B 0,C 180,E1 -21360.127,E2 -21360.127} C_VEL
LIN {X 0,Y 217.827,Z 325.01,A -85,B 0,C 180,E1 -21361.621,E2 -21361.621} C_VEL
LIN {X 0,Y 220.007,Z 312.604,A -85,B 0,C 180,E1 -21362.756,E2 -21362.756} C_VEL
LIN {X 0,Y 221.732,Z 299.36,A -85,B 0,C 180,E1 -21363.581,E2 -21363.581} C_VEL
LIN {X 0,Y 222.734,Z 283.604,A -85,B 0,C 180,E1 -21364.159,E2 -21364.159} C_VEL
LIN {X 0,Y 224.441,Z 242.365,A -85,B 0,C 180,E1 -21365.434,E2 -21365.434} C_VEL
LIN {X 0,Y 222.783,Z 230.737,A -85,B 0,C 180,E1 -21366.189,E2 -21366.189} C_VEL
LIN {X 0,Y 216.068,Z 214.573,A -85,B 0,C 180,E1 -21368.158,E2 -21368.158} C_VEL
LIN {X 0,Y 210.33,Z 202.893,A -85,B 0,C 180,E1 -21369.895,E2 -21369.895} C_VEL
LIN {X 0,Y 205.741,Z 194.529,A -85,B 0,C 180,E1 -21371.343,E2 -21371.343} C_VEL
LIN {X 0,Y 203.124,Z 190.048,A -85,B 0,C 180,E1 -21372.2,E2 -21372.2} C_VEL
LIN {X 0,Y 200.897,Z 185.866,A -85,B 0,C 180,E1 -21373.054,E2 -21373.054} C_VEL
LIN {X 0,Y 199.572,Z 181.126,A -85,B 0,C 180,E1 -21376.06,E2 -21376.06} C_VEL
LIN {X 0,Y 199.61,Z 181.12,A -85,B 0,C 180,E1 -21380.768,E2 -21380.768} C_VEL
LIN {X 0,Y 199.611,Z 181.12,A -85,B 0,C 180,E1 -21385.713,E2 -21385.713} C_VEL
LIN {X 0,Y 199.686,Z 181.111,A -85,B 0,C 180,E1 -21388.134,E2 -21388.134} C_VEL
LIN {X 0,Y 199.644,Z 181.109,A -85,B 0,C 180,E1 -21392.765,E2 -21392.765} C_VEL
LIN {X 0,Y 199.71,Z 181.099,A -85,B 0,C 180,E1 -21397.226,E2 -21397.226} C_VEL
LIN {X 0,Y 199.797,Z 181.088,A -85,B 0,C 180,E1 -21401.758,E2 -21401.758} C_VEL
LIN {X 0,Y 199.837,Z 181.09,A -85,B 0,C 180,E1 -21405.748,E2 -21405.748} C_VEL
LIN {X 0,Y 200.023,Z 181.069,A -85,B 0,C 180,E1 -21409.882,E2 -21409.882} C_VEL
LIN {X 0,Y 200.024,Z 181.058,A -85,B 0,C 180,E1 -21413.949,E2 -21413.949} C_VEL
LIN {X 0,Y 200.322,Z 181.027,A -85,B 0,C 180,E1 -21417.99,E2 -21417.99} C_VEL
LIN {X 0,Y 200.477,Z 181.002,A -85,B 0,C 180,E1 -21420,E2 -21420} C_VEL
LIN {X 0,Y 200.027,Z 181.065,A -85,B 0,C 180,E1 -21424.03,E2 -21424.03} C_VEL
LIN {X 0,Y 200.09,Z 181.06,A -85,B 0,C 180,E1 -21428.077,E2 -21428.077} C_VEL
LIN {X 0,Y 199.875,Z 181.076,A -85,B 0,C 180,E1 -21432.179,E2 -21432.179} C_VEL
LIN {X 0,Y 199.807,Z 181.089,A -85,B 0,C 180,E1 -21436.343,E2 -21436.343} C_VEL
LIN {X 0,Y 199.825,Z 181.087,A -85,B 0,C 180,E1 -21438.454,E2 -21438.454} C_VEL
LIN {X 0,Y 199.738,Z 181.1,A -85,B 0,C 180,E1 -21443.817,E2 -21443.817} C_VEL
LIN {X 0,Y 199.714,Z 181.1,A -85,B 0,C 180,E1 -21448.387,E2 -21448.387} C_VEL
LIN {X 0,Y 199.665,Z 181.107,A -85,B 0,C 180,E1 -21452.352,E2 -21452.352} C_VEL
LIN {X 0,Y 199.641,Z 181.114,A -85,B 0,C 180,E1 -21456.76,E2 -21456.76} C_VEL
LIN {X 0,Y 199.64,Z 181.112,A -85,B 0,C 180,E1 -21459.321,E2 -21459.321} C_VEL
LIN {X 0,Y 199.581,Z 181.12,A -85,B 0,C 180,E1 -21464.771,E2 -21464.771} C_VEL
LIN {X 0,Y 199.58,Z 181.124,A -85,B 0,C 180,E1 -21466.773,E2 -21466.773} C_VEL
LIN {X 0,Y 200.696,Z 184.153,A -85,B 0,C 180,E1 -21467.257,E2 -21467.257} C_VEL
LIN {X 0,Y 202.607,Z 186.399,A -85,B 0,C 180,E1 -21467.863,E2 -21467.863} C_VEL
LIN {X 0,Y 204.809,Z 189.776,A -85,B 0,C 180,E1 -21468.577,E2 -21468.577} C_VEL
LIN {X 0,Y 211.328,Z 200.079,A -85,B 0,C 180,E1 -21470.575,E2 -21470.575} C_VEL
LIN {X 0,Y 217.334,Z 211.95,A -85,B 0,C 180,E1 -21472.361,E2 -21472.361} C_VEL
LIN {X 0,Y 223.699,Z 226.48,A -85,B 0,C 180,E1 -21474.183,E2 -21474.183} C_VEL
LIN {X 0,Y 225.073,Z 229.94,A -85,B 0,C 180,E1 -21474.57,E2 -21474.57} C_VEL
LIN {X 0,Y 222.559,Z 284.525,A -85,B 0,C 180,E1 -21476.242,E2 -21476.242} C_VEL
LIN {X 0,Y 221.388,Z 297.582,A -85,B 0,C 180,E1 -21476.908,E2 -21476.908} C_VEL
LIN {X 0,Y 219.658,Z 309.862,A -85,B 0,C 180,E1 -21477.865,E2 -21477.865} C_VEL
LIN {X 0,Y 217.55,Z 321.691,A -85,B 0,C 180,E1 -21479.146,E2 -21479.146} C_VEL
LIN {X 0,Y 215.135,Z 332.432,A -85,B 0,C 180,E1 -21480.658,E2 -21480.658} C_VEL
LIN {X 0,Y 212.236,Z 343.379,A -85,B 0,C 180,E1 -21482.648,E2 -21482.648} C_VEL
LIN {X 0,Y 209.491,Z 353.125,A -85,B 0,C 180,E1 -21484.931,E2 -21484.931} C_VEL
LIN {X 0,Y 206.815,Z 361.909,A -85,B 0,C 180,E1 -21487.524,E2 -21487.524} C_VEL
LIN {X 0,Y 204.037,Z 369.598,A -85,B 0,C 180,E1 -21490.377,E2 -21490.377} C_VEL
LIN {X 0,Y 202.17,Z 374.846,A -85,B 0,C 180,E1 -21492.813,E2 -21492.813} C_VEL
LIN {X 0,Y 200.369,Z 379.934,A -85,B 0,C 180,E1 -21495.787,E2 -21495.787} C_VEL
LIN {X 0,Y 199.021,Z 383.883,A -85,B 0,C 180,E1 -21498.801,E2 -21498.801} C_VEL
LIN {X 0,Y 198.154,Z 386.797,A -85,B 0,C 180,E1 -21501.844,E2 -21501.844} C_VEL
LIN {X 0,Y 197.6,Z 388.691,A -85,B 0,C 180,E1 -21504.795,E2 -21504.795} C_VEL
LIN {X 0,Y 197.361,Z 389.79,A -85,B 0,C 180,E1 -21507.959,E2 -21507.959} C_VEL
LIN {X 0,Y 197.329,Z 390.018,A -85,B 0,C 180,E1 -21510,E2 -21510} C_VEL
LIN {X 0,Y 197.36,Z 389.824,A -85,B 0,C 180,E1 -21512.041,E2 -21512.041} C_VEL
LIN {X 0,Y 197.722,Z 388.269,A -85,B 0,C 180,E1 -21516.121,E2 -21516.121} C_VEL
LIN {X 0,Y 198.078,Z 386.911,A -85,B 0,C 180,E1 -21518.159,E2 -21518.159} C_VEL
LIN {X 0,Y 198.991,Z 384.038,A -85,B 0,C 180,E1 -21521.201,E2 -21521.201} C_VEL
LIN {X 0,Y 200.339,Z 380.142,A -85,B 0,C 180,E1 -21524.215,E2 -21524.215} C_VEL
LIN {X 0,Y 202.122,Z 375.116,A -85,B 0,C 180,E1 -21527.191,E2 -21527.191} C_VEL
LIN {X 0,Y 204.406,Z 368.783,A -85,B 0,C 180,E1 -21530.11,E2 -21530.11} C_VEL
LIN {X 0,Y 207.199,Z 360.857,A -85,B 0,C 180,E1 -21532.959,E2 -21532.959} C_VEL
LIN {X 0,Y 209.605,Z 352.836,A -85,B 0,C 180,E1 -21535.293,E2 -21535.293} C_VEL
LIN {X 0,Y 212.521,Z 342.924,A -85,B 0,C 180,E1 -21537.579,E2 -21537.579} C_VEL
LIN {X 0,Y 215.104,Z 333.216,A -85,B 0,C 180,E1 -21539.346,E2 -21539.346} C_VEL
LIN {X 0,Y 217.462,Z 322.698,A -85,B 0,C 180,E1 -21540.867,E2 -21540.867} C_VEL
LIN {X 0,Y 219.779,Z 310.031,A -85,B 0,C 180,E1 -21542.25,E2 -21542.25} C_VEL
LIN {X 0,Y 221.427,Z 297.644,A -85,B 0,C 180,E1 -21543.236,E2 -21543.236} C_VEL
LIN {X 0,Y 222.689,Z 284.418,A -85,B 0,C 180,E1 -21543.896,E2 -21543.896} C_VEL
LIN {X 0,Y 225.193,Z 230.22,A -85,B 0,C 180,E1 -21545.554,E2 -21545.554} C_VEL
LIN {X 0,Y 219.312,Z 216.092,A -85,B 0,C 180,E1 -21547.233,E2 -21547.233} C_VEL
LIN {X 0,Y 212.689,Z 202.592,A -85,B 0,C 180,E1 -21549.183,E2 -21549.183} C_VEL
LIN {X 0,Y 209.047,Z 196.331,A -85,B 0,C 180,E1 -21550.282,E2 -21550.282} C_VEL
LIN {X 0,Y 204.527,Z 189.454,A -85,B 0,C 180,E1 -21551.686,E2 -21551.686} C_VEL
LIN {X 0,Y 201.966,Z 185.608,A -85,B 0,C 180,E1 -21552.521,E2 -21552.521} C_VEL
LIN {X 0,Y 200.1,Z 183.056,A -85,B 0,C 180,E1 -21553.139,E2 -21553.139} C_VEL
LIN {X 0,Y 199.577,Z 181.126,A -85,B 0,C 180,E1 -21553.391,E2 -21553.391} C_VEL
LIN {X 0,Y 199.583,Z 181.117,A -85,B 0,C 180,E1 -21558.005,E2 -21558.005} C_VEL
LIN {X 0,Y 199.642,Z 181.113,A -85,B 0,C 180,E1 -21560.756,E2 -21560.756} C_VEL
LIN {X 0,Y 199.634,Z 181.108,A -85,B 0,C 180,E1 -21565.718,E2 -21565.718} C_VEL
LIN {X 0,Y 199.704,Z 181.103,A -85,B 0,C 180,E1 -21568.137,E2 -21568.137} C_VEL
LIN {X 0,Y 199.687,Z 181.1,A -85,B 0,C 180,E1 -21572.772,E2 -21572.772} C_VEL
LIN {X 0,Y 199.738,Z 181.092,A -85,B 0,C 180,E1 -21577.229,E2 -21577.229} C_VEL
LIN {X 0,Y 199.797,Z 181.096,A -85,B 0,C 180,E1 -21581.757,E2 -21581.757} C_VEL
LIN {X 0,Y 199.848,Z 181.079,A -85,B 0,C 180,E1 -21585.749,E2 -21585.749} C_VEL
LIN {X 0,Y 200.07,Z 181.055,A -85,B 0,C 180,E1 -21589.884,E2 -21589.884} C_VEL
LIN {X 0,Y 200.034,Z 181.066,A -85,B 0,C 180,E1 -21593.95,E2 -21593.95} C_VEL
LIN {X 0,Y 200.322,Z 181.016,A -85,B 0,C 180,E1 -21597.989,E2 -21597.989} C_VEL
LIN {X 0,Y 200.476,Z 181,A -85,B 0,C 180,E1 -21600,E2 -21600} C_VEL
LIN {X 0,Y 200.031,Z 181.063,A -85,B 0,C 180,E1 -21604.029,E2 -21604.029} C_VEL
LIN {X 0,Y 200.111,Z 181.051,A -85,B 0,C 180,E1 -21608.076,E2 -21608.076} C_VEL
LIN {X 0,Y 199.887,Z 181.071,A -85,B 0,C 180,E1 -21612.179,E2 -21612.179} C_VEL
LIN {X 0,Y 199.805,Z 181.096,A -85,B 0,C 180,E1 -21616.343,E2 -21616.343} C_VEL
LIN {X 0,Y 199.682,Z 181.1,A -85,B 0,C 180,E1 -21620.607,E2 -21620.607} C_VEL
LIN {X 0,Y 199.664,Z 181.101,A -85,B 0,C 180,E1 -21624.986,E2 -21624.986} C_VEL
LIN {X 0,Y 199.664,Z 181.106,A -85,B 0,C 180,E1 -21629.524,E2 -21629.524} C_VEL
LIN {X 0,Y 199.671,Z 181.114,A -85,B 0,C 180,E1 -21632.356,E2 -21632.356} C_VEL
LIN {X 0,Y 199.623,Z 181.119,A -85,B 0,C 180,E1 -21636.763,E2 -21636.763} C_VEL
LIN {X 0,Y 199.608,Z 181.118,A -85,B 0,C 180,E1 -21639.328,E2 -21639.328} C_VEL
LIN {X 0,Y 199.605,Z 181.255,A -85,B 0,C 180,E1 -21643.931,E2 -21643.931} C_VEL
LIN {X 0,Y 201.03,Z 186.271,A -85,B 0,C 180,E1 -21646.988,E2 -21646.988} C_VEL
LIN {X 0,Y 203.61,Z 190.665,A -85,B 0,C 180,E1 -21647.863,E2 -21647.863} C_VEL
LIN {X 0,Y 210.375,Z 202.914,A -85,B 0,C 180,E1 -21650.036,E2 -21650.036} C_VEL
LIN {X 0,Y 213.423,Z 208.813,A -85,B 0,C 180,E1 -21650.965,E2 -21650.965} C_VEL
LIN {X 0,Y 215.268,Z 213.958,A -85,B 0,C 180,E1 -21651.575,E2 -21651.575} C_VEL
LIN {X 0,Y 216.418,Z 219.519,A -85,B 0,C 180,E1 -21652.044,E2 -21652.044} C_VEL
LIN {X 0,Y 218.259,Z 239.067,A -85,B 0,C 180,E1 -21653.208,E2 -21653.208} C_VEL
LIN {X 0,Y 218.798,Z 244.307,A -85,B 0,C 180,E1 -21653.522,E2 -21653.522} C_VEL
LIN {X 0,Y 216.304,Z 294.742,A -85,B 0,C 180,E1 -21655.114,E2 -21655.114} C_VEL
LIN {X 0,Y 214.859,Z 308.148,A -85,B 0,C 180,E1 -21655.861,E2 -21655.861} C_VEL
LIN {X 0,Y 212.838,Z 320.237,A -85,B 0,C 180,E1 -21656.846,E2 -21656.846} C_VEL
LIN {X 0,Y 210.375,Z 332.423,A -85,B 0,C 180,E1 -21658.254,E2 -21658.254} C_VEL
LIN {X 0,Y 207.408,Z 343.976,A -85,B 0,C 180,E1 -21660.013,E2 -21660.013} C_VEL
LIN {X 0,Y 204.369,Z 354.382,A -85,B 0,C 180,E1 -21662.06,E2 -21662.06} C_VEL
LIN {X 0,Y 201.617,Z 362.89,A -85,B 0,C 180,E1 -21664.169,E2 -21664.169} C_VEL
LIN {X 0,Y 198.889,Z 371.171,A -85,B 0,C 180,E1 -21666.743,E2 -21666.743} C_VEL
LIN {X 0,Y 196.293,Z 378.415,A -85,B 0,C 180,E1 -21669.569,E2 -21669.569} C_VEL
LIN {X 0,Y 193.741,Z 385.494,A -85,B 0,C 180,E1 -21673.13,E2 -21673.13} C_VEL
LIN {X 0,Y 192.077,Z 390.203,A -85,B 0,C 180,E1 -21676.242,E2 -21676.242} C_VEL
LIN {X 0,Y 191.021,Z 393.804,A -85,B 0,C 180,E1 -21679.4,E2 -21679.4} C_VEL
LIN {X 0,Y 190.532,Z 395.661,A -85,B 0,C 180,E1 -21681.515,E2 -21681.515} C_VEL
LIN {X 0,Y 190.127,Z 398.051,A -85,B 0,C 180,E1 -21685.76,E2 -21685.76} C_VEL
LIN {X 0,Y 190.141,Z 398.659,A -85,B 0,C 180,E1 -21687.882,E2 -21687.882} C_VEL
LIN {X 0,Y 190.202,Z 398.871,A -85,B 0,C 180,E1 -21690,E2 -21690} C_VEL
LIN {X 0,Y 190.116,Z 398.302,A -85,B 0,C 180,E1 -21693.525,E2 -21693.525} C_VEL
LIN {X 0,Y 190.276,Z 397.025,A -85,B 0,C 180,E1 -21696.362,E2 -21696.362} C_VEL
LIN {X 0,Y 190.532,Z 395.618,A -85,B 0,C 180,E1 -21698.485,E2 -21698.485} C_VEL
LIN {X 0,Y 191.307,Z 392.67,A -85,B 0,C 180,E1 -21701.657,E2 -21701.657} C_VEL
LIN {X 0,Y 192.52,Z 388.684,A -85,B 0,C 180,E1 -21704.805,E2 -21704.805} C_VEL
LIN {X 0,Y 194.791,Z 382.564,A -85,B 0,C 180,E1 -21708.403,E2 -21708.403} C_VEL
LIN {X 0,Y 197.189,Z 375.944,A -85,B 0,C 180,E1 -21711.399,E2 -21711.399} C_VEL
LIN {X 0,Y 199.903,Z 367.737,A -85,B 0,C 180,E1 -21714.344,E2 -21714.344} C_VEL
LIN {X 0,Y 202.75,Z 359.086,A -85,B 0,C 180,E1 -21716.784,E2 -21716.784} C_VEL
LIN {X 0,Y 205.993,Z 348.585,A -85,B 0,C 180,E1 -21719.09,E2 -21719.09} C_VEL
LIN {X 0,Y 209.18,Z 336.762,A -85,B 0,C 180,E1 -21721.102,E2 -21721.102} C_VEL
LIN {X 0,Y 211.822,Z 324.842,A -85,B 0,C 180,E1 -21722.626,E2 -21722.626} C_VEL
LIN {X 0,Y 214.07,Z 312.434,A -85,B 0,C 180,E1 -21723.784,E2 -21723.784} C_VEL
LIN {X 0,Y 215.783,Z 299.839,A -85,B 0,C 180,E1 -21724.591,E2 -21724.591} C_VEL
LIN {X 0,Y 216.801,Z 285.428,A -85,B 0,C 180,E1 -21725.151,E2 -21725.151} C_VEL
LIN {X 0,Y 218.665,Z 243.381,A -85,B 0,C 180,E1 -21726.47,E2 -21726.47} C_VEL
LIN {X 0,Y 217.326,Z 233.673,A -85,B 0,C 180,E1 -21727.122,E2 -21727.122} C_VEL
LIN {X 0,Y 211.081,Z 218.302,A -85,B 0,C 180,E1 -21729.063,E2 -21729.063} C_VEL
LIN {X 0,Y 205.337,Z 206.529,A -85,B 0,C 180,E1 -21730.897,E2 -21730.897} C_VEL
LIN {X 0,Y 201.262,Z 198.974,A -85,B 0,C 180,E1 -21732.258,E2 -21732.258} C_VEL
LIN {X 0,Y 196.166,Z 190.296,A -85,B 0,C 180,E1 -21734.047,E2 -21734.047} C_VEL
LIN {X 0,Y 193.544,Z 185.664,A -85,B 0,C 180,E1 -21735.104,E2 -21735.104} C_VEL
LIN {X 0,Y 192.536,Z 182.002,A -85,B 0,C 180,E1 -21737.65,E2 -21737.65} C_VEL
LIN {X 0,Y 192.587,Z 181.996,A -85,B 0,C 180,E1 -21743.402,E2 -21743.402} C_VEL
LIN {X 0,Y 192.605,Z 181.993,A -85,B 0,C 180,E1 -21747.061,E2 -21747.061} C_VEL
LIN {X 0,Y 192.621,Z 181.988,A -85,B 0,C 180,E1 -21751.685,E2 -21751.685} C_VEL
LIN {X 0,Y 192.68,Z 181.978,A -85,B 0,C 180,E1 -21756.345,E2 -21756.345} C_VEL
LIN {X 0,Y 192.732,Z 181.969,A -85,B 0,C 180,E1 -21761.458,E2 -21761.458} C_VEL
LIN {X 0,Y 192.765,Z 181.974,A -85,B 0,C 180,E1 -21765.214,E2 -21765.214} C_VEL
LIN {X 0,Y 192.946,Z 181.948,A -85,B 0,C 180,E1 -21769.567,E2 -21769.567} C_VEL
LIN {X 0,Y 192.986,Z 181.934,A -85,B 0,C 180,E1 -21773.728,E2 -21773.728} C_VEL
LIN {X 0,Y 193.264,Z 181.906,A -85,B 0,C 180,E1 -21777.916,E2 -21777.916} C_VEL
LIN {X 0,Y 193.441,Z 181.877,A -85,B 0,C 180,E1 -21780,E2 -21780} C_VEL
LIN {X 0,Y 192.973,Z 181.941,A -85,B 0,C 180,E1 -21784.177,E2 -21784.177} C_VEL
LIN {X 0,Y 193.037,Z 181.939,A -85,B 0,C 180,E1 -21788.374,E2 -21788.374} C_VEL
LIN {X 0,Y 192.803,Z 181.959,A -85,B 0,C 180,E1 -21792.633,E2 -21792.633} C_VEL
LIN {X 0,Y 192.772,Z 181.961,A -85,B 0,C 180,E1 -21796.958,E2 -21796.958} C_VEL
LIN {X 0,Y 192.643,Z 181.984,A -85,B 0,C 180,E1 -21801.397,E2 -21801.397} C_VEL
LIN {X 0,Y 192.665,Z 181.982,A -85,B 0,C 180,E1 -21804.225,E2 -21804.225} C_VEL
LIN {X 0,Y 192.651,Z 181.984,A -85,B 0,C 180,E1 -21808.892,E2 -21808.892} C_VEL
LIN {X 0,Y 192.602,Z 181.991,A -85,B 0,C 180,E1 -21813.186,E2 -21813.186} C_VEL
LIN {X 0,Y 192.575,Z 181.995,A -85,B 0,C 180,E1 -21818.347,E2 -21818.347} C_VEL
LIN {X 0,Y 192.494,Z 182.003,A -85,B 0,C 180,E1 -21823.097,E2 -21823.097} C_VEL
LIN {X 0,Y 192.537,Z 182.004,A -85,B 0,C 180,E1 -21824.843,E2 -21824.843} C_VEL
LIN {X 0,Y 193.462,Z 184.67,A -85,B 0,C 180,E1 -21825.257,E2 -21825.257} C_VEL
LIN {X 0,Y 195.767,Z 187.5,A -85,B 0,C 180,E1 -21826.068,E2 -21826.068} C_VEL
LIN {X 0,Y 197.883,Z 190.767,A -85,B 0,C 180,E1 -21826.819,E2 -21826.819} C_VEL
LIN {X 0,Y 203.648,Z 199.414,A -85,B 0,C 180,E1 -21828.732,E2 -21828.732} C_VEL
LIN {X 0,Y 208.167,Z 207.139,A -85,B 0,C 180,E1 -21830.163,E2 -21830.163} C_VEL
LIN {X 0,Y 215.351,Z 222.335,A -85,B 0,C 180,E1 -21832.381,E2 -21832.381} C_VEL
LIN {X 0,Y 219.251,Z 231.955,A -85,B 0,C 180,E1 -21833.553,E2 -21833.553} C_VEL
LIN {X 0,Y 216.621,Z 285.881,A -85,B 0,C 180,E1 -21835.243,E2 -21835.243} C_VEL
LIN {X 0,Y 215.289,Z 299.121,A -85,B 0,C 180,E1 -21835.97,E2 -21835.97} C_VEL
LIN {X 0,Y 213.312,Z 312.287,A -85,B 0,C 180,E1 -21837.069,E2 -21837.069} C_VEL
LIN {X 0,Y 211.126,Z 323.591,A -85,B 0,C 180,E1 -21838.38,E2 -21838.38} C_VEL
LIN {X 0,Y 208.279,Z 335.227,A -85,B 0,C 180,E1 -21840.151,E2 -21840.151} C_VEL
LIN {X 0,Y 205.334,Z 345.677,A -85,B 0,C 180,E1 -21842.203,E2 -21842.203} C_VEL
LIN {X 0,Y 202.6,Z 354.815,A -85,B 0,C 180,E1 -21844.491,E2 -21844.491} C_VEL
LIN {X 0,Y 199.702,Z 363.461,A -85,B 0,C 180,E1 -21847.225,E2 -21847.225} C_VEL
LIN {X 0,Y 196.918,Z 370.873,A -85,B 0,C 180,E1 -21850.181,E2 -21850.181} C_VEL
LIN {X 0,Y 194.706,Z 376.818,A -85,B 0,C 180,E1 -21853.216,E2 -21853.216} C_VEL
LIN {X 0,Y 192.929,Z 381.515,A -85,B 0,C 180,E1 -21856.303,E2 -21856.303} C_VEL
LIN {X 0,Y 191.681,Z 385.107,A -85,B 0,C 180,E1 -21859.436,E2 -21859.436} C_VEL
LIN {X 0,Y 191.116,Z 386.96,A -85,B 0,C 180,E1 -21861.541,E2 -21861.541} C_VEL
LIN {X 0,Y 190.497,Z 389.03,A -85,B 0,C 180,E1 -21864.948,E2 -21864.948} C_VEL
LIN {X 0,Y 190.272,Z 389.952,A -85,B 0,C 180,E1 -21867.883,E2 -21867.883} C_VEL
LIN {X 0,Y 190.237,Z 390.18,A -85,B 0,C 180,E1 -21870,E2 -21870} C_VEL
LIN {X 0,Y 190.271,Z 389.986,A -85,B 0,C 180,E1 -21872.117,E2 -21872.117} C_VEL
LIN {X 0,Y 190.46,Z 389.14,A -85,B 0,C 180,E1 -21874.924,E2 -21874.924} C_VEL
LIN {X 0,Y 191.062,Z 387.072,A -85,B 0,C 180,E1 -21878.461,E2 -21878.461} C_VEL
LIN {X 0,Y 192.011,Z 384.2,A -85,B 0,C 180,E1 -21881.613,E2 -21881.613} C_VEL
LIN {X 0,Y 193.441,Z 380.304,A -85,B 0,C 180,E1 -21884.733,E2 -21884.733} C_VEL
LIN {X 0,Y 195.324,Z 375.277,A -85,B 0,C 180,E1 -21887.809,E2 -21887.809} C_VEL
LIN {X 0,Y 197.752,Z 368.943,A -85,B 0,C 180,E1 -21890.817,E2 -21890.817} C_VEL
LIN {X 0,Y 200.657,Z 361.017,A -85,B 0,C 180,E1 -21893.752,E2 -21893.752} C_VEL
LIN {X 0,Y 203.282,Z 352.751,A -85,B 0,C 180,E1 -21896.214,E2 -21896.214} C_VEL
LIN {X 0,Y 206.246,Z 343.083,A -85,B 0,C 180,E1 -21898.493,E2 -21898.493} C_VEL
LIN {X 0,Y 208.946,Z 333.374,A -85,B 0,C 180,E1 -21900.3,E2 -21900.3} C_VEL
LIN {X 0,Y 211.402,Z 322.854,A -85,B 0,C 180,E1 -21901.854,E2 -21901.854} C_VEL
LIN {X 0,Y 213.826,Z 310.185,A -85,B 0,C 180,E1 -21903.263,E2 -21903.263} C_VEL
LIN {X 0,Y 215.579,Z 297.427,A -85,B 0,C 180,E1 -21904.294,E2 -21904.294} C_VEL
LIN {X 0,Y 216.831,Z 284.603,A -85,B 0,C 180,E1 -21904.94,E2 -21904.94} C_VEL
LIN {X 0,Y 219.383,Z 232.065,A -85,B 0,C 180,E1 -21906.578,E2 -21906.578} C_VEL
LIN {X 0,Y 212.909,Z 216.824,A -85,B 0,C 180,E1 -21908.53,E2 -21908.53} C_VEL
LIN {X 0,Y 206.43,Z 203.812,A -85,B 0,C 180,E1 -21910.566,E2 -21910.566} C_VEL
LIN {X 0,Y 200.311,Z 194.34,A -85,B 0,C 180,E1 -21912.541,E2 -21912.541} C_VEL
LIN {X 0,Y 197.451,Z 190.236,A -85,B 0,C 180,E1 -21913.512,E2 -21913.512} C_VEL
LIN {X 0,Y 195.245,Z 186.75,A -85,B 0,C 180,E1 -21914.309,E2 -21914.309} C_VEL
LIN {X 0,Y 193.283,Z 184.399,A -85,B 0,C 180,E1 -21915.003,E2 -21915.003} C_VEL
LIN {X 0,Y 192.533,Z 181.998,A -85,B 0,C 180,E1 -21915.406,E2 -21915.406} C_VEL
LIN {X 0,Y 192.542,Z 182.001,A -85,B 0,C 180,E1 -21920.042,E2 -21920.042} C_VEL
LIN {X 0,Y 192.599,Z 181.993,A -85,B 0,C 180,E1 -21924.278,E2 -21924.278} C_VEL
LIN {X 0,Y 192.608,Z 181.992,A -85,B 0,C 180,E1 -21929.28,E2 -21929.28} C_VEL
LIN {X 0,Y 192.665,Z 181.972,A -85,B 0,C 180,E1 -21931.692,E2 -21931.692} C_VEL
LIN {X 0,Y 192.706,Z 181.974,A -85,B 0,C 180,E1 -21936.348,E2 -21936.348} C_VEL
LIN {X 0,Y 192.732,Z 181.977,A -85,B 0,C 180,E1 -21941.457,E2 -21941.457} C_VEL
LIN {X 0,Y 192.772,Z 181.956,A -85,B 0,C 180,E1 -21945.214,E2 -21945.214} C_VEL
LIN {X 0,Y 192.981,Z 181.94,A -85,B 0,C 180,E1 -21949.508,E2 -21949.508} C_VEL
LIN {X 0,Y 193.062,Z 181.917,A -85,B 0,C 180,E1 -21951.627,E2 -21951.627} C_VEL
LIN {X 0,Y 193.264,Z 181.895,A -85,B 0,C 180,E1 -21957.916,E2 -21957.916} C_VEL
LIN {X 0,Y 193.441,Z 181.875,A -85,B 0,C 180,E1 -21960,E2 -21960} C_VEL
LIN {X 0,Y 192.977,Z 181.939,A -85,B 0,C 180,E1 -21964.177,E2 -21964.177} C_VEL
LIN {X 0,Y 193.062,Z 181.931,A -85,B 0,C 180,E1 -21968.373,E2 -21968.373} C_VEL
LIN {X 0,Y 192.81,Z 181.949,A -85,B 0,C 180,E1 -21972.633,E2 -21972.633} C_VEL
LIN {X 0,Y 192.757,Z 181.972,A -85,B 0,C 180,E1 -21976.959,E2 -21976.959} C_VEL
LIN {X 0,Y 192.617,Z 181.988,A -85,B 0,C 180,E1 -21981.4,E2 -21981.4} C_VEL
LIN {X 0,Y 192.647,Z 181.978,A -85,B 0,C 180,E1 -21984.213,E2 -21984.213} C_VEL
LIN {X 0,Y 192.644,Z 181.985,A -85,B 0,C 180,E1 -21988.889,E2 -21988.889} C_VEL
LIN {X 0,Y 192.596,Z 181.992,A -85,B 0,C 180,E1 -21993.186,E2 -21993.186} C_VEL
LIN {X 0,Y 192.551,Z 181.993,A -85,B 0,C 180,E1 -21998.352,E2 -21998.352} C_VEL
LIN {X 0,Y 192.538,Z 182.091,A -85,B 0,C 180,E1 -22002.36,E2 -22002.36} C_VEL
LIN {X 0,Y 193.585,Z 185.83,A -85,B 0,C 180,E1 -22004.884,E2 -22004.884} C_VEL
LIN {X 0,Y 196.178,Z 190.279,A -85,B 0,C 180,E1 -22005.858,E2 -22005.858} C_VEL
LIN {X 0,Y 201.063,Z 198.637,A -85,B 0,C 180,E1 -22007.584,E2 -22007.584} C_VEL
LIN {X 0,Y 206.985,Z 209.588,A -85,B 0,C 180,E1 -22009.547,E2 -22009.547} C_VEL
LIN {X 0,Y 213.064,Z 222.763,A -85,B 0,C 180,E1 -22011.478,E2 -22011.478} C_VEL
LIN {X 0,Y 217.581,Z 234.37,A -85,B 0,C 180,E1 -22012.885,E2 -22012.885} C_VEL
LIN {X 0,Y 218.259,Z 239.067,A -85,B 0,C 180,E1 -22013.208,E2 -22013.208} C_VEL
LIN {X 0,Y 218.128,Z 242.305,A -85,B 0,C 180,E1 -22013.312,E2 -22013.312} C_VEL
LIN {X 0,Y 216.776,Z 246.76,A -85,B 0,C 180,E1 -22013.227,E2 -22013.227} C_VEL
LIN {X 0,Y 213.083,Z 255.502,A -85,B 0,C 180,E1 -22012.848,E2 -22012.848} C_VEL
LIN {X 0,Y 212.354,Z 259.49,A -85,B 0,C 180,E1 -22012.865,E2 -22012.865} C_VEL
LIN {X 0,Y 210.444,Z 295.566,A -85,B 0,C 180,E1 -22014.057,E2 -22014.057} C_VEL
LIN {X 0,Y 208.911,Z 308.776,A -85,B 0,C 180,E1 -22014.823,E2 -22014.823} C_VEL
LIN {X 0,Y 206.728,Z 321.187,A -85,B 0,C 180,E1 -22015.88,E2 -22015.88} C_VEL
LIN {X 0,Y 203.981,Z 333.849,A -85,B 0,C 180,E1 -22017.429,E2 -22017.429} C_VEL
LIN {X 0,Y 200.949,Z 345.112,A -85,B 0,C 180,E1 -22019.237,E2 -22019.237} C_VEL
LIN {X 0,Y 197.768,Z 355.256,A -85,B 0,C 180,E1 -22021.332,E2 -22021.332} C_VEL
LIN {X 0,Y 194.636,Z 364.398,A -85,B 0,C 180,E1 -22023.748,E2 -22023.748} C_VEL
LIN {X 0,Y 191.66,Z 372.996,A -85,B 0,C 180,E1 -22026.65,E2 -22026.65} C_VEL
LIN {X 0,Y 188.821,Z 380.489,A -85,B 0,C 180,E1 -22029.862,E2 -22029.862} C_VEL
LIN {X 0,Y 186.248,Z 387.022,A -85,B 0,C 180,E1 -22033.56,E2 -22033.56} C_VEL
LIN {X 0,Y 184.734,Z 391.349,A -85,B 0,C 180,E1 -22036.805,E2 -22036.805} C_VEL
LIN {X 0,Y 184.031,Z 393.642,A -85,B 0,C 180,E1 -22038.992,E2 -22038.992} C_VEL
LIN {X 0,Y 183.504,Z 395.499,A -85,B 0,C 180,E1 -22041.188,E2 -22041.188} C_VEL
LIN {X 0,Y 183.034,Z 397.888,A -85,B 0,C 180,E1 -22045.596,E2 -22045.596} C_VEL
LIN {X 0,Y 183.041,Z 398.497,A -85,B 0,C 180,E1 -22047.8,E2 -22047.8} C_VEL
LIN {X 0,Y 183.111,Z 398.709,A -85,B 0,C 180,E1 -22050,E2 -22050} C_VEL
LIN {X 0,Y 183.032,Z 398.24,A -85,B 0,C 180,E1 -22053.301,E2 -22053.301} C_VEL
LIN {X 0,Y 183.209,Z 396.862,A -85,B 0,C 180,E1 -22056.608,E2 -22056.608} C_VEL
LIN {X 0,Y 183.504,Z 395.455,A -85,B 0,C 180,E1 -22058.812,E2 -22058.812} C_VEL
LIN {X 0,Y 184.339,Z 392.506,A -85,B 0,C 180,E1 -22062.104,E2 -22062.104} C_VEL
LIN {X 0,Y 185.63,Z 388.52,A -85,B 0,C 180,E1 -22065.368,E2 -22065.368} C_VEL
LIN {X 0,Y 188.049,Z 382.399,A -85,B 0,C 180,E1 -22069.088,E2 -22069.088} C_VEL
LIN {X 0,Y 190.582,Z 375.793,A -85,B 0,C 180,E1 -22072.174,E2 -22072.174} C_VEL
LIN {X 0,Y 193.49,Z 367.423,A -85,B 0,C 180,E1 -22075.264,E2 -22075.264} C_VEL
LIN {X 0,Y 196.431,Z 358.921,A -85,B 0,C 180,E1 -22077.718,E2 -22077.718} C_VEL
LIN {X 0,Y 199.808,Z 348.419,A -85,B 0,C 180,E1 -22080.081,E2 -22080.081} C_VEL
LIN {X 0,Y 203.121,Z 336.595,A -85,B 0,C 180,E1 -22082.139,E2 -22082.139} C_VEL
LIN {X 0,Y 205.887,Z 324.674,A -85,B 0,C 180,E1 -22083.69,E2 -22083.69} C_VEL
LIN {X 0,Y 208.223,Z 312.264,A -85,B 0,C 180,E1 -22084.867,E2 -22084.867} C_VEL
LIN {X 0,Y 209.995,Z 299.554,A -85,B 0,C 180,E1 -22085.696,E2 -22085.696} C_VEL
LIN {X 0,Y 211.055,Z 285.098,A -85,B 0,C 180,E1 -22086.262,E2 -22086.262} C_VEL
LIN {X 0,Y 212.893,Z 243.84,A -85,B 0,C 180,E1 -22087.6,E2 -22087.6} C_VEL
LIN {X 0,Y 211.849,Z 236.349,A -85,B 0,C 180,E1 -22088.132,E2 -22088.132} C_VEL
LIN {X 0,Y 205.873,Z 221.479,A -85,B 0,C 180,E1 -22090.1,E2 -22090.1} C_VEL
LIN {X 0,Y 199.602,Z 208.471,A -85,B 0,C 180,E1 -22092.237,E2 -22092.237} C_VEL
LIN {X 0,Y 194.004,Z 198.494,A -85,B 0,C 180,E1 -22094.248,E2 -22094.248} C_VEL
LIN {X 0,Y 191.33,Z 194.04,A -85,B 0,C 180,E1 -22095.26,E2 -22095.26} C_VEL
LIN {X 0,Y 188.899,Z 190.087,A -85,B 0,C 180,E1 -22096.216,E2 -22096.216} C_VEL
LIN {X 0,Y 186.272,Z 185.725,A -85,B 0,C 180,E1 -22097.302,E2 -22097.302} C_VEL
LIN {X 0,Y 185.463,Z 182.883,A -85,B 0,C 180,E1 -22099.372,E2 -22099.372} C_VEL
LIN {X 0,Y 185.506,Z 182.877,A -85,B 0,C 180,E1 -22102.711,E2 -22102.711} C_VEL
LIN {X 0,Y 185.531,Z 182.874,A -85,B 0,C 180,E1 -22107.972,E2 -22107.972} C_VEL
LIN {X 0,Y 185.547,Z 182.873,A -85,B 0,C 180,E1 -22110.595,E2 -22110.595} C_VEL
LIN {X 0,Y 185.58,Z 182.869,A -85,B 0,C 180,E1 -22115.382,E2 -22115.382} C_VEL
LIN {X 0,Y 185.675,Z 182.85,A -85,B 0,C 180,E1 -22121.134,E2 -22121.134} C_VEL
LIN {X 0,Y 185.696,Z 182.854,A -85,B 0,C 180,E1 -22124.637,E2 -22124.637} C_VEL
LIN {X 0,Y 185.889,Z 182.826,A -85,B 0,C 180,E1 -22129.418,E2 -22129.418} C_VEL
LIN {X 0,Y 185.949,Z 182.81,A -85,B 0,C 180,E1 -22133.49,E2 -22133.49} C_VEL
LIN {X 0,Y 186.208,Z 182.785,A -85,B 0,C 180,E1 -22137.837,E2 -22137.837} C_VEL
LIN {X 0,Y 186.405,Z 182.753,A -85,B 0,C 180,E1 -22140,E2 -22140} C_VEL
LIN {X 0,Y 185.919,Z 182.818,A -85,B 0,C 180,E1 -22144.336,E2 -22144.336} C_VEL
LIN {X 0,Y 185.984,Z 182.819,A -85,B 0,C 180,E1 -22148.694,E2 -22148.694} C_VEL
LIN {X 0,Y 185.73,Z 182.843,A -85,B 0,C 180,E1 -22153.123,E2 -22153.123} C_VEL
LIN {X 0,Y 185.718,Z 182.839,A -85,B 0,C 180,E1 -22157.622,E2 -22157.622} C_VEL
LIN {X 0,Y 185.601,Z 182.856,A -85,B 0,C 180,E1 -22162.251,E2 -22162.251} C_VEL
LIN {X 0,Y 185.564,Z 182.861,A -85,B 0,C 180,E1 -22167.032,E2 -22167.032} C_VEL
LIN {X 0,Y 185.58,Z 182.868,A -85,B 0,C 180,E1 -22169.493,E2 -22169.493} C_VEL
LIN {X 0,Y 185.512,Z 182.875,A -85,B 0,C 180,E1 -22174.63,E2 -22174.63} C_VEL
LIN {X 0,Y 185.545,Z 182.873,A -85,B 0,C 180,E1 -22177.304,E2 -22177.304} C_VEL
